FUNCTION_BLOCK "Side_Shifters"   // FB12, LAD
{ S7_Optimized_Access := 'TRUE' }
// stored: MemoryReserve 100, SetENOAutomatically false
   VAR_INPUT
      set_Hydraulic_Up { ExternalAccessible := 'False'; ExternalVisible := 'False'; ExternalWritable := 'False'} : Bool;
      set_Hydraulic_Down { ExternalAccessible := 'False'; ExternalVisible := 'False'; ExternalWritable := 'False'} : Bool;
      set_SL_Hydraulic_Up : Bool;
      set_SL_Hydraulic_Down : Bool;
      set_SR_Hydraulic_Up : Bool;
      set_SR_Hydraulic_Down : Bool;
      set_SL_Hydraulic_Unit : Bool;
      set_SR_Hydraulic_Unit : Bool;
      set_Go_To_ST1 : Bool;
      set_Go_To_ST2 : Bool;
      set_Go_To_ST3 : Bool;
      set_Go_To_ST4 : Bool;
      ST1_Empty : Bool;
      ST2_Empty : Bool;
      ST3_Empty : Bool;
      ST4_Empty : Bool;
      Homing_1_SR : Int;
      Homing_2_SR : Int;
      Homing_3_SR : Int;
      Homing_4_SR : Int;
      Homing_1_SL : Int;
      Homing_2_SL : Int;
      Homing_3_SL : Int;
      Homing_4_SL : Int;
      SL_Drive_Forward : Bool;
      SL_Drive_Backward : Bool;
      SR_Drive_Forward : Bool;
      SR_Drive_Backward : Bool;
      iSL_Sen_Drv_1 : Bool;
      iSL_Sen_Drv_2 : Bool;
      iSL_Sen_Drv_3 : Bool;
      iSL_Sen_Drv_4 : Bool;
      iSR_Sen_Drv_1 : Bool;
      iSR_Sen_Drv_2 : Bool;
      iSR_Sen_Drv_3 : Bool;
      iSR_Sen_Drv_4 : Bool;
      iSL_Sen_Val1_Up : Bool;
      iSL_Sen_Val1_Down : Bool;
      iSL_Sen_Val2_Up : Bool;
      iSL_Sen_Val2_Down : Bool;
      iSR_Sen_Val1_Up : Bool;
      iSR_Sen_Val1_Down : Bool;
      iSR_Sen_Val2_Up : Bool;
      iSR_Sen_Val2_Down : Bool;
      iSL_Distance : Int;
      iSR_Correct : Int;
      iSR_Distance : Int;
      iSL_Hydraulic_Filtr : Bool;
      iSR_Hydraulic_Empty : Bool;
      HWIdentSL : HW_IO;
      HWIdentSR : HW_IO;
      Reset_Drive : Bool;
      Reset_Hydro : Bool;
   END_VAR
   VAR_OUTPUT
      oSL_Valve_Up { ExternalAccessible := 'False'; ExternalVisible := 'False'; ExternalWritable := 'False'} : Bool;
      oSL_Valve_Down { ExternalAccessible := 'False'; ExternalVisible := 'False'; ExternalWritable := 'False'} : Bool;
      oSL_Hydraulic_Unit { ExternalAccessible := 'False'; ExternalVisible := 'False'; ExternalWritable := 'False'} : Bool;
      oSR_Valve_Up { ExternalAccessible := 'False'; ExternalVisible := 'False'; ExternalWritable := 'False'} : Bool;
      oSR_Valve_Down { ExternalAccessible := 'False'; ExternalVisible := 'False'; ExternalWritable := 'False'} : Bool;
      oSR_Hydraulic_Unit { ExternalAccessible := 'False'; ExternalVisible := 'False'; ExternalWritable := 'False'} : Bool;
      oHydraulic_Status_LED_UP_1 : Bool;
      oHydraulic_Status_LED_UP_2 : Bool;
      oHydraulic_Status_LED_DOWN_1 : Bool;
      oHydraulic_Status_LED_DOWN_2 : Bool;
      oSL_Communication_OK : Bool;
      oSR_Communication_OK : Bool;
      oSL_Forward_Flag : Bool;
      oSL_Backward_Flag : Bool;
      oSR_Forward_Flag : Bool;
      oSR_Backward_Flag : Bool;
      oST1_1_Move_Flag : Bool;
      oST1_2_Move_Flag : Bool;
      oST2_1_Move_Flag : Bool;
      oST2_2_Move_Flag : Bool;
      oST3_1_Move_flag : Bool;
      oST3_2_Move_Flag : Bool;
      oST4_1_Move_Flag : Bool;
      oST4_2_Move_Flag : Bool;
   END_VAR
   VAR_IN_OUT
      iSL_Drive_Param : "SEW_MOVIKIT_VelocityDrive_STATUS_V2.1";
      iSR_Drive_Param : "SEW_MOVIKIT_VelocityDrive_STATUS_V2.1";
      oSL_Drive_Param : "SEW_MOVIKIT_VelocityDrive_SETPOINTS_V2.1";
      oSR_Drive_Param : "SEW_MOVIKIT_VelocityDrive_SETPOINTS_V2.1";
   END_VAR
   VAR
      Hydraulic_SL { ExternalAccessible := 'False'; ExternalVisible := 'False'; ExternalWritable := 'False'} : "Side_Hydraulic";
      Hydraulic_SR { ExternalAccessible := 'False'; ExternalVisible := 'False'; ExternalWritable := 'False'} : "Side_Hydraulic";
      Side_Driver_Instance { S7_SetPoint := 'True'} : "Side_Driver";
      Side_Shifter_Auto_Instance { S7_SetPoint := 'True'} : "Side_Shifter_Auto";
      SL_Auto_Speed { S7_SetPoint := 'True'} : Int := 1000;
      SR_Auto_Speed { S7_SetPoint := 'True'} : Int := 1000;
      SL_Auto_Forward : Bool;
      SL_Auto_Backward : Bool;
      SR_Auto_Forward : Bool;
      SR_Auto_Backward : Bool;
      SR_Distance_Correct : Int;
      SL_Error_Laser : Bool;
      SR_Error_Laser : Bool;
      SL_SR_InPosition : Bool;
      SL_Sen_Up : Bool;
      SL_Sen_Down : Bool;
      SR_Sen_Up : Bool;
      SR_Sen_Down : Bool;
      SL_Error_Hyd : Bool;
      SR_Error_Hyd : Bool;
      Error_Drive : Bool;
      Error_Hydro : Bool;
      Status_Sen_Up : Bool;
      Status_Sen_Down : Bool;
      RL_Speed : Int;
      RR_Speed : Int;
      Step_Move_Pallets : Int;
      Row_Start : Int;
      Row_Destination : Int;
      Column_Start : Int;
      Column_Destination : Int;
      TON_iSR_Error { S7_SetPoint := 'True'} : TON_TIME;
      TON_iSL_Error { S7_SetPoint := 'True'} : TON_TIME;
   END_VAR
   VAR_TEMP
      i : SInt;
      FoundIndex : SInt;
   END_VAR
BEGIN

REGION Network 1: Hydraulic control SL
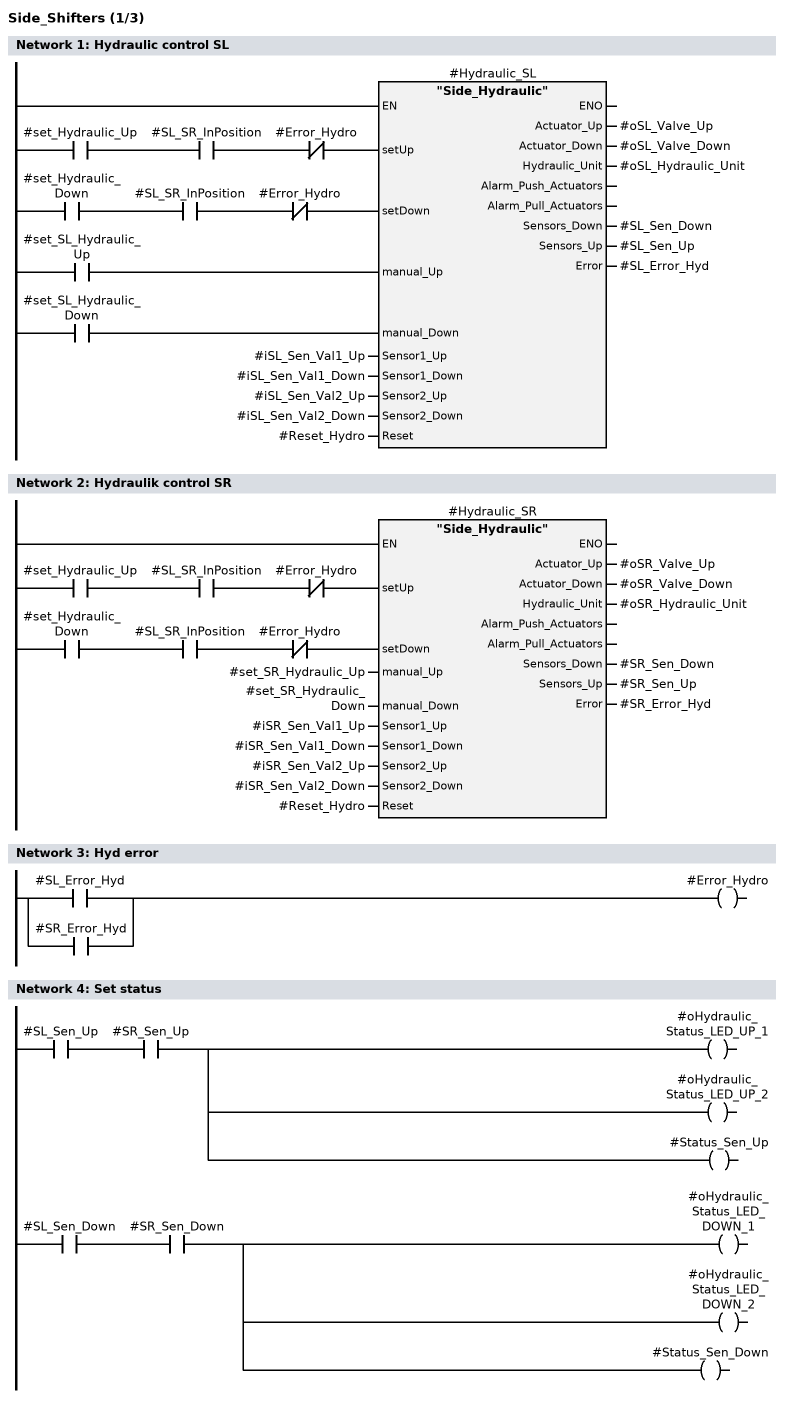
   RUNG wire#powerrail
      #Hydraulic_SL(setUp := wire#w1, setDown := wire#w2, manual_Up := wire#w3, manual_Down := wire#w4, Sensor1_Up := #iSL_Sen_Val1_Up, Sensor1_Down := #iSL_Sen_Val1_Down, Sensor2_Up := #iSL_Sen_Val2_Up, Sensor2_Down := #iSL_Sen_Val2_Down, Reset := #Reset_Hydro, Actuator_Up => #oSL_Valve_Up, Actuator_Down => #oSL_Valve_Down, Hydraulic_Unit => #oSL_Hydraulic_Unit, Alarm_Push_Actuators =>, Alarm_Pull_Actuators =>, Sensors_Down => #SL_Sen_Down, Sensors_Up => #SL_Sen_Up, Error => #SL_Error_Hyd)
   END_RUNG
   RUNG wire#powerrail
      Contact( #set_Hydraulic_Up )
      Contact( #SL_SR_InPosition )
      I_Contact( #Error_Hydro )
   END_RUNG wire#w1
   RUNG wire#powerrail
      Contact( #set_Hydraulic_Down )
      Contact( #SL_SR_InPosition )
      I_Contact( #Error_Hydro )
   END_RUNG wire#w2
   RUNG wire#powerrail
      Contact( #set_SL_Hydraulic_Up )
   END_RUNG wire#w3
   RUNG wire#powerrail
      Contact( #set_SL_Hydraulic_Down )
   END_RUNG wire#w4
   // the same network as SCL:
   #Hydraulic_SL(setUp := #set_Hydraulic_Up AND #SL_SR_InPosition AND NOT #Error_Hydro,   // "Side_Hydraulic"
                 setDown := #set_Hydraulic_Down AND #SL_SR_InPosition AND NOT #Error_Hydro,
                 manual_Up := #set_SL_Hydraulic_Up,
                 manual_Down := #set_SL_Hydraulic_Down,
                 Sensor1_Up := #iSL_Sen_Val1_Up,
                 Sensor1_Down := #iSL_Sen_Val1_Down,
                 Sensor2_Up := #iSL_Sen_Val2_Up,
                 Sensor2_Down := #iSL_Sen_Val2_Down,
                 Reset := #Reset_Hydro,
                 Actuator_Up => #oSL_Valve_Up,
                 Actuator_Down => #oSL_Valve_Down,
                 Hydraulic_Unit => #oSL_Hydraulic_Unit,
                 Sensors_Down => #SL_Sen_Down,
                 Sensors_Up => #SL_Sen_Up,
                 Error => #SL_Error_Hyd);
END_REGION

REGION Network 2: Hydraulik control SR
   RUNG wire#powerrail
      #Hydraulic_SR(setUp := wire#w1, setDown := wire#w2, manual_Up := #set_SR_Hydraulic_Up, manual_Down := #set_SR_Hydraulic_Down, Sensor1_Up := #iSR_Sen_Val1_Up, Sensor1_Down := #iSR_Sen_Val1_Down, Sensor2_Up := #iSR_Sen_Val2_Up, Sensor2_Down := #iSR_Sen_Val2_Down, Reset := #Reset_Hydro, Actuator_Up => #oSR_Valve_Up, Actuator_Down => #oSR_Valve_Down, Hydraulic_Unit => #oSR_Hydraulic_Unit, Alarm_Push_Actuators =>, Alarm_Pull_Actuators =>, Sensors_Down => #SR_Sen_Down, Sensors_Up => #SR_Sen_Up, Error => #SR_Error_Hyd)
   END_RUNG
   RUNG wire#powerrail
      Contact( #set_Hydraulic_Up )
      Contact( #SL_SR_InPosition )
      I_Contact( #Error_Hydro )
   END_RUNG wire#w1
   RUNG wire#powerrail
      Contact( #set_Hydraulic_Down )
      Contact( #SL_SR_InPosition )
      I_Contact( #Error_Hydro )
   END_RUNG wire#w2
   // the same network as SCL:
   #Hydraulic_SR(setUp := #set_Hydraulic_Up AND #SL_SR_InPosition AND NOT #Error_Hydro,   // "Side_Hydraulic"
                 setDown := #set_Hydraulic_Down AND #SL_SR_InPosition AND NOT #Error_Hydro,
                 manual_Up := #set_SR_Hydraulic_Up,
                 manual_Down := #set_SR_Hydraulic_Down,
                 Sensor1_Up := #iSR_Sen_Val1_Up,
                 Sensor1_Down := #iSR_Sen_Val1_Down,
                 Sensor2_Up := #iSR_Sen_Val2_Up,
                 Sensor2_Down := #iSR_Sen_Val2_Down,
                 Reset := #Reset_Hydro,
                 Actuator_Up => #oSR_Valve_Up,
                 Actuator_Down => #oSR_Valve_Down,
                 Hydraulic_Unit => #oSR_Hydraulic_Unit,
                 Sensors_Down => #SR_Sen_Down,
                 Sensors_Up => #SR_Sen_Up,
                 Error => #SR_Error_Hyd);
END_REGION

REGION Network 3: Hyd error
   RUNG wire#powerrail
      Contact( #SL_Error_Hyd )
      wire#w1
      Coil( #Error_Hydro )
   END_RUNG
   RUNG wire#powerrail
      Contact( #SR_Error_Hyd )
   END_RUNG wire#w1
   // the same network as SCL:
   #Error_Hydro := #SL_Error_Hyd OR #SR_Error_Hyd;
END_REGION

REGION Network 4: Set status
   RUNG wire#powerrail
      Contact( #SL_Sen_Up )
      Contact( #SR_Sen_Up )
      wire#w1
      Coil( #oHydraulic_Status_LED_UP_1 )
   END_RUNG
   RUNG wire#w1
      Coil( #oHydraulic_Status_LED_UP_2 )
   END_RUNG
   RUNG wire#w1
      Coil( #Status_Sen_Up )
   END_RUNG
   RUNG wire#powerrail
      Contact( #SL_Sen_Down )
      Contact( #SR_Sen_Down )
      wire#w2
      Coil( #oHydraulic_Status_LED_DOWN_1 )
   END_RUNG
   RUNG wire#w2
      Coil( #oHydraulic_Status_LED_DOWN_2 )
   END_RUNG
   RUNG wire#w2
      Coil( #Status_Sen_Down )
   END_RUNG
   // the same network as SCL:
   #oHydraulic_Status_LED_UP_1 := #SL_Sen_Up AND #SR_Sen_Up;
   #oHydraulic_Status_LED_UP_2 := #oHydraulic_Status_LED_UP_1;
   #Status_Sen_Up := #oHydraulic_Status_LED_UP_1;
   #oHydraulic_Status_LED_DOWN_1 := #SL_Sen_Down AND #SR_Sen_Down;
   #oHydraulic_Status_LED_DOWN_2 := #oHydraulic_Status_LED_DOWN_1;
   #Status_Sen_Down := #oHydraulic_Status_LED_DOWN_1;
END_REGION

REGION Network 5: Make correct on SR distance
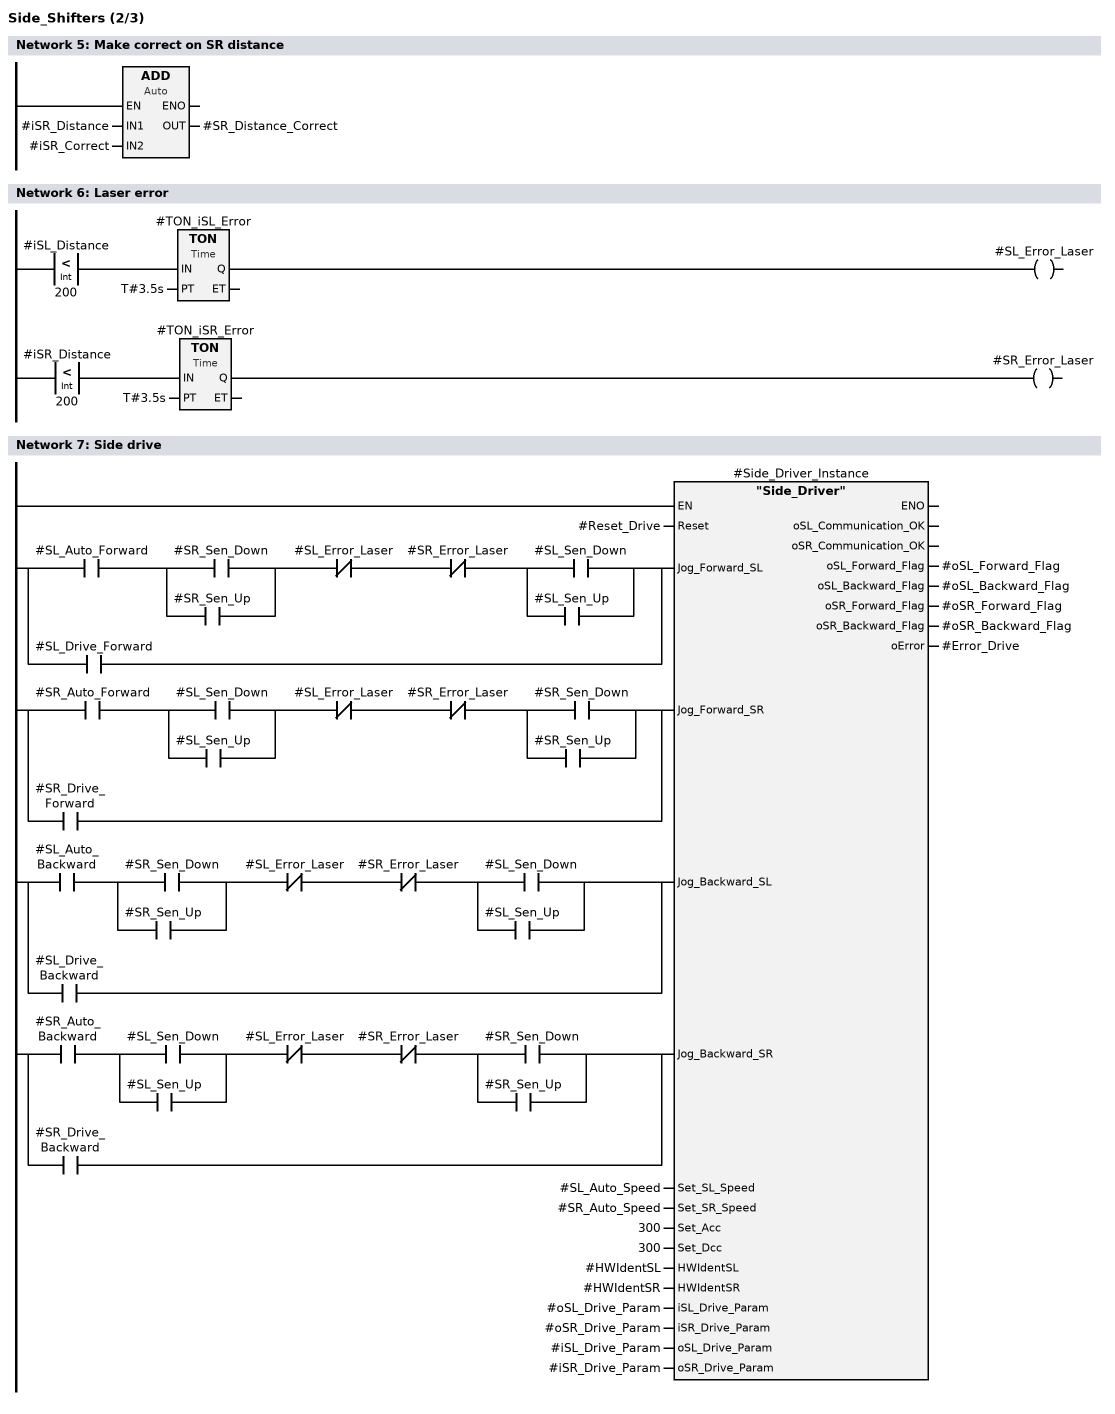
   RUNG wire#powerrail
      Add(in1 := #iSR_Distance, in2 := #iSR_Correct, out => #SR_Distance_Correct)
   END_RUNG
   // the same network as SCL:
   #SR_Distance_Correct := #iSR_Distance + #iSR_Correct;
END_REGION

REGION Network 6: Laser error
   RUNG wire#powerrail
      { S7_Templates := "SrcType := Int" } LT_Contact(in1 := #iSL_Distance, in2 := 200)
      { S7_Templates := "time_type := Time" } #TON_iSL_Error.TON(pt := T#3.5s, et =>)
      Coil( #SL_Error_Laser )
   END_RUNG
   RUNG wire#powerrail
      { S7_Templates := "SrcType := Int" } LT_Contact(in1 := #iSR_Distance, in2 := 200)
      { S7_Templates := "time_type := Time" } #TON_iSR_Error.TON(pt := T#3.5s, et =>)
      Coil( #SR_Error_Laser )
   END_RUNG
   // the same network as SCL:
   #TON_iSL_Error(IN := #iSL_Distance < 200, PT := T#3.5s);   // TON
   #SL_Error_Laser := #TON_iSL_Error.Q;
   #TON_iSR_Error(IN := #iSR_Distance < 200, PT := T#3.5s);   // TON
   #SR_Error_Laser := #TON_iSR_Error.Q;
END_REGION

REGION Network 7: Side drive
   RUNG wire#powerrail
      #Side_Driver_Instance(Jog_Forward_SL := wire#w4, Jog_Forward_SR := wire#w8, Jog_Backward_SL := wire#w12, Jog_Backward_SR := wire#w16, Reset := #Reset_Drive, Set_SL_Speed := #SL_Auto_Speed, Set_SR_Speed := #SR_Auto_Speed, Set_Acc := 300, Set_Dcc := 300, HWIdentSL := #HWIdentSL, HWIdentSR := #HWIdentSR, iSL_Drive_Param := #oSL_Drive_Param, iSR_Drive_Param := #oSR_Drive_Param, oSL_Drive_Param := #iSL_Drive_Param, oSR_Drive_Param := #iSR_Drive_Param, oSL_Communication_OK =>, oSR_Communication_OK =>, oSL_Forward_Flag => #oSL_Forward_Flag, oSL_Backward_Flag => #oSL_Backward_Flag, oSR_Forward_Flag => #oSR_Forward_Flag, oSR_Backward_Flag => #oSR_Backward_Flag, oError => #Error_Drive)
   END_RUNG
   RUNG wire#powerrail
      Contact( #SL_Auto_Forward )
      wire#w1
      Contact( #SR_Sen_Down )
      wire#w2
      I_Contact( #SL_Error_Laser )
      I_Contact( #SR_Error_Laser )
      wire#w3
      Contact( #SL_Sen_Down )
   END_RUNG wire#w4
   RUNG wire#w1
      Contact( #SR_Sen_Up )
   END_RUNG wire#w2
   RUNG wire#w3
      Contact( #SL_Sen_Up )
   END_RUNG wire#w4
   RUNG wire#powerrail
      Contact( #SL_Drive_Forward )
   END_RUNG wire#w4
   RUNG wire#powerrail
      Contact( #SR_Auto_Forward )
      wire#w5
      Contact( #SL_Sen_Down )
      wire#w6
      I_Contact( #SL_Error_Laser )
      I_Contact( #SR_Error_Laser )
      wire#w7
      Contact( #SR_Sen_Down )
   END_RUNG wire#w8
   RUNG wire#w5
      Contact( #SL_Sen_Up )
   END_RUNG wire#w6
   RUNG wire#w7
      Contact( #SR_Sen_Up )
   END_RUNG wire#w8
   RUNG wire#powerrail
      Contact( #SR_Drive_Forward )
   END_RUNG wire#w8
   RUNG wire#powerrail
      Contact( #SL_Auto_Backward )
      wire#w9
      Contact( #SR_Sen_Down )
      wire#w10
      I_Contact( #SL_Error_Laser )
      I_Contact( #SR_Error_Laser )
      wire#w11
      Contact( #SL_Sen_Down )
   END_RUNG wire#w12
   RUNG wire#w9
      Contact( #SR_Sen_Up )
   END_RUNG wire#w10
   RUNG wire#w11
      Contact( #SL_Sen_Up )
   END_RUNG wire#w12
   RUNG wire#powerrail
      Contact( #SL_Drive_Backward )
   END_RUNG wire#w12
   RUNG wire#powerrail
      Contact( #SR_Auto_Backward )
      wire#w13
      Contact( #SL_Sen_Down )
      wire#w14
      I_Contact( #SL_Error_Laser )
      I_Contact( #SR_Error_Laser )
      wire#w15
      Contact( #SR_Sen_Down )
   END_RUNG wire#w16
   RUNG wire#w13
      Contact( #SL_Sen_Up )
   END_RUNG wire#w14
   RUNG wire#w15
      Contact( #SR_Sen_Up )
   END_RUNG wire#w16
   RUNG wire#powerrail
      Contact( #SR_Drive_Backward )
   END_RUNG wire#w16
   // the same network as SCL:
   #Side_Driver_Instance(Reset := #Reset_Drive,   // "Side_Driver"
                         Jog_Forward_SL := (#SL_Auto_Forward AND (#SR_Sen_Down OR #SR_Sen_Up) AND NOT #SL_Error_Laser AND NOT #SR_Error_Laser AND (#SL_Sen_Down OR #SL_Sen_Up)) OR #SL_Drive_Forward,
                         Jog_Forward_SR := (#SR_Auto_Forward AND (#SL_Sen_Down OR #SL_Sen_Up) AND NOT #SL_Error_Laser AND NOT #SR_Error_Laser AND (#SR_Sen_Down OR #SR_Sen_Up)) OR #SR_Drive_Forward,
                         Jog_Backward_SL := (#SL_Auto_Backward AND (#SR_Sen_Down OR #SR_Sen_Up) AND NOT #SL_Error_Laser AND NOT #SR_Error_Laser AND (#SL_Sen_Down OR #SL_Sen_Up)) OR #SL_Drive_Backward,
                         Jog_Backward_SR := (#SR_Auto_Backward AND (#SL_Sen_Down OR #SL_Sen_Up) AND NOT #SL_Error_Laser AND NOT #SR_Error_Laser AND (#SR_Sen_Down OR #SR_Sen_Up)) OR #SR_Drive_Backward,
                         Set_SL_Speed := #SL_Auto_Speed,
                         Set_SR_Speed := #SR_Auto_Speed,
                         Set_Acc := 300,
                         Set_Dcc := 300,
                         HWIdentSL := #HWIdentSL,
                         HWIdentSR := #HWIdentSR,
                         iSL_Drive_Param := #oSL_Drive_Param,
                         iSR_Drive_Param := #oSR_Drive_Param,
                         oSL_Drive_Param := #iSL_Drive_Param,
                         oSR_Drive_Param := #iSR_Drive_Param,
                         oSL_Forward_Flag => #oSL_Forward_Flag,
                         oSL_Backward_Flag => #oSL_Backward_Flag,
                         oSR_Forward_Flag => #oSR_Forward_Flag,
                         oSR_Backward_Flag => #oSR_Backward_Flag,
                         oError => #Error_Drive);
END_REGION

REGION Network 8: Auto moving
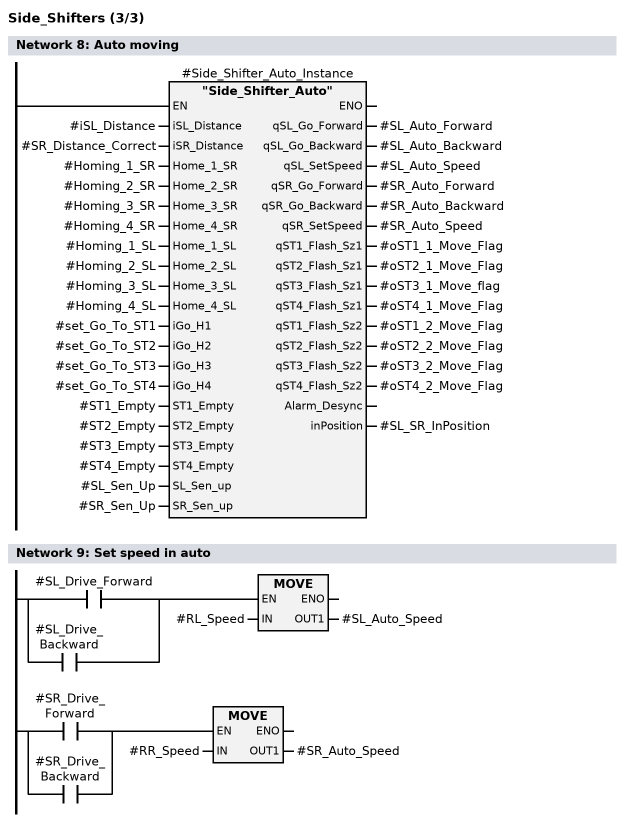
   RUNG wire#powerrail
      #Side_Shifter_Auto_Instance(iSL_Distance := #iSL_Distance, iSR_Distance := #SR_Distance_Correct, Home_1_SR := #Homing_1_SR, Home_2_SR := #Homing_2_SR, Home_3_SR := #Homing_3_SR, Home_4_SR := #Homing_4_SR, Home_1_SL := #Homing_1_SL, Home_2_SL := #Homing_2_SL, Home_3_SL := #Homing_3_SL, Home_4_SL := #Homing_4_SL, iGo_H1 := #set_Go_To_ST1, iGo_H2 := #set_Go_To_ST2, iGo_H3 := #set_Go_To_ST3, iGo_H4 := #set_Go_To_ST4, ST1_Empty := #ST1_Empty, ST2_Empty := #ST2_Empty, ST3_Empty := #ST3_Empty, ST4_Empty := #ST4_Empty, SL_Sen_up := #SL_Sen_Up, SR_Sen_up := #SR_Sen_Up, qSL_Go_Forward => #SL_Auto_Forward, qSL_Go_Backward => #SL_Auto_Backward, qSL_SetSpeed => #SL_Auto_Speed, qSR_Go_Forward => #SR_Auto_Forward, qSR_Go_Backward => #SR_Auto_Backward, qSR_SetSpeed => #SR_Auto_Speed, qST1_Flash_Sz1 => #oST1_1_Move_Flag, qST2_Flash_Sz1 => #oST2_1_Move_Flag, qST3_Flash_Sz1 => #oST3_1_Move_flag, qST4_Flash_Sz1 => #oST4_1_Move_Flag, qST1_Flash_Sz2 => #oST1_2_Move_Flag, qST2_Flash_Sz2 => #oST2_2_Move_Flag, qST3_Flash_Sz2 => #oST3_2_Move_Flag, qST4_Flash_Sz2 => #oST4_2_Move_Flag, Alarm_Desync =>, inPosition => #SL_SR_InPosition)
   END_RUNG
   // the same network as SCL:
   #Side_Shifter_Auto_Instance(iSL_Distance := #iSL_Distance,   // "Side_Shifter_Auto"
                           iSR_Distance := #SR_Distance_Correct,
                           Home_1_SR := #Homing_1_SR,
                           Home_2_SR := #Homing_2_SR,
                           Home_3_SR := #Homing_3_SR,
                           Home_4_SR := #Homing_4_SR,
                           Home_1_SL := #Homing_1_SL,
                           Home_2_SL := #Homing_2_SL,
                           Home_3_SL := #Homing_3_SL,
                           Home_4_SL := #Homing_4_SL,
                           iGo_H1 := #set_Go_To_ST1,
                           iGo_H2 := #set_Go_To_ST2,
                           iGo_H3 := #set_Go_To_ST3,
                           iGo_H4 := #set_Go_To_ST4,
                           ST1_Empty := #ST1_Empty,
                           ST2_Empty := #ST2_Empty,
                           ST3_Empty := #ST3_Empty,
                           ST4_Empty := #ST4_Empty,
                           SL_Sen_up := #SL_Sen_Up,
                           SR_Sen_up := #SR_Sen_Up,
                           qSL_Go_Forward => #SL_Auto_Forward,
                           qSL_Go_Backward => #SL_Auto_Backward,
                           qSL_SetSpeed => #SL_Auto_Speed,
                           qSR_Go_Forward => #SR_Auto_Forward,
                           qSR_Go_Backward => #SR_Auto_Backward,
                           qSR_SetSpeed => #SR_Auto_Speed,
                           qST1_Flash_Sz1 => #oST1_1_Move_Flag,
                           qST2_Flash_Sz1 => #oST2_1_Move_Flag,
                           qST3_Flash_Sz1 => #oST3_1_Move_flag,
                           qST4_Flash_Sz1 => #oST4_1_Move_Flag,
                           qST1_Flash_Sz2 => #oST1_2_Move_Flag,
                           qST2_Flash_Sz2 => #oST2_2_Move_Flag,
                           qST3_Flash_Sz2 => #oST3_2_Move_Flag,
                           qST4_Flash_Sz2 => #oST4_2_Move_Flag,
                           inPosition => #SL_SR_InPosition);
END_REGION

REGION Network 9: Set speed in auto
   RUNG wire#powerrail
      Contact( #SL_Drive_Forward )
      wire#w1
      Move(in := #RL_Speed, out1 => #SL_Auto_Speed)
   END_RUNG
   RUNG wire#powerrail
      Contact( #SL_Drive_Backward )
   END_RUNG wire#w1
   RUNG wire#powerrail
      Contact( #SR_Drive_Forward )
      wire#w2
      Move(in := #RR_Speed, out1 => #SR_Auto_Speed)
   END_RUNG
   RUNG wire#powerrail
      Contact( #SR_Drive_Backward )
   END_RUNG wire#w2
   // the same network as SCL:
   IF #SL_Drive_Forward OR #SL_Drive_Backward THEN #SL_Auto_Speed := #RL_Speed; END_IF;
   IF #SR_Drive_Forward OR #SR_Drive_Backward THEN #SR_Auto_Speed := #RR_Speed; END_IF;
END_REGION

REGION Network 10 (SCL): SS1 - Move Pallet
   IF #HWIdentSL = "S1R1M~Module_I_O_(05_words)_1" THEN

       IF (#Hydraulic_SL.Actuator_Up OR #Hydraulic_SR.Actuator_Up) AND #Status_Sen_Up AND #Step_Move_Pallets = 0 THEN
           #Step_Move_Pallets := 1;
           IF #oST1_1_Move_Flag THEN
               #Row_Start := 1;
               #Column_Start := 11;
           ELSIF #oST2_1_Move_Flag THEN
               #Row_Start := 2;
               #Column_Start := 12;
           ELSIF #oST3_1_Move_flag THEN
               #Row_Start := 3;
               #Column_Start := 11;
           ELSIF #oST4_1_Move_Flag THEN
               #Row_Start := 4;
               #Column_Start := 11;
           END_IF;

       ELSIF (#Hydraulic_SL.Actuator_Down OR #Hydraulic_SR.Actuator_Down) AND #Status_Sen_Up AND #Step_Move_Pallets = 1 THEN
           #Step_Move_Pallets := 2;
           IF #oST1_1_Move_Flag THEN
               #Row_Destination := 1;
               #Column_Destination := 11;
           ELSIF #oST2_1_Move_Flag THEN
               #Row_Destination := 2;
               #Column_Destination := 12;
           ELSIF #oST3_1_Move_flag THEN
               #Row_Destination := 3;
               #Column_Destination := 11;
           ELSIF #oST4_1_Move_Flag THEN
               #Row_Destination := 4;
               #Column_Destination := 11;
           END_IF;

       ELSIF #Step_Move_Pallets = 2 THEN
           FOR #i := 1 TO 24 DO
               IF ("Pallets_Stations".Pallets[#i].Station_Current_Position[1] = #Row_Start) AND
                   ("Pallets_Stations".Pallets[#i].Station_Current_Position[2] = #Column_Start) THEN
                   #FoundIndex := #i;
                   EXIT;
               END_IF;
           END_FOR;

           IF #FoundIndex <> 0 THEN
               "Pallets_Stations".Pallets[#FoundIndex].Station_Current_Position[1] := #Row_Destination;
               "Pallets_Stations".Pallets[#FoundIndex].Station_Current_Position[2] := #Column_Destination;
           END_IF;
           #Step_Move_Pallets := 0;

       END_IF;
   END_IF;
END_REGION

REGION Network 11 (SCL): SS2 - Move Pallet
   IF #HWIdentSL = "S2R2M~Module_I_O_(05_words)_1" THEN
       #Column_Start := 1;
       IF (#Hydraulic_SL.Actuator_Up OR #Hydraulic_SR.Actuator_Up) AND #Status_Sen_Up AND #Step_Move_Pallets = 0 THEN
           #Step_Move_Pallets := 1;
           IF #oST1_1_Move_Flag THEN
               #Row_Start := 1;
           ELSIF #oST2_1_Move_Flag THEN
               #Row_Start := 2;
           ELSIF #oST3_1_Move_flag THEN
               #Row_Start := 3;
           ELSIF #oST4_1_Move_Flag THEN
               #Row_Start := 4;
           END_IF;

       ELSIF (#Hydraulic_SL.Actuator_Down OR #Hydraulic_SR.Actuator_Down) AND #Status_Sen_Up AND #Step_Move_Pallets = 1 THEN
           #Step_Move_Pallets := 2;
           IF #oST1_1_Move_Flag THEN
               #Row_Destination := 1;
           ELSIF #oST2_1_Move_Flag THEN
               #Row_Destination := 2;
           ELSIF #oST3_1_Move_flag THEN
               #Row_Destination := 3;
           ELSIF #oST4_1_Move_Flag THEN
               #Row_Destination := 4;
           END_IF;

       ELSIF #Step_Move_Pallets = 2 THEN
           FOR #i := 1 TO 24 DO
               IF ("Pallets_Stations".Pallets[#i].Station_Current_Position[1] = #Row_Start) AND
                   ("Pallets_Stations".Pallets[#i].Station_Current_Position[2] = #Column_Start) THEN
                   #FoundIndex := #i;
                   EXIT;
               END_IF;
           END_FOR;

           IF #FoundIndex <> 0 THEN
               "Pallets_Stations".Pallets[#FoundIndex].Station_Current_Position[1] := #Row_Destination;
               "Pallets_Stations".Pallets[#FoundIndex].Station_Current_Position[2] := #Column_Destination;
           END_IF;
           #Step_Move_Pallets := 0;

       END_IF;
   END_IF;
END_REGION
END_FUNCTION_BLOCK

FUNCTION_BLOCK "Side_Shifter_Auto"   // FB13, LAD
{ S7_Optimized_Access := 'TRUE' }
// stored: MemoryReserve 100, SetENOAutomatically false
   VAR_INPUT
      iSL_Distance : Int;
      iSR_Distance : Int;
      Home_1_SR : Int;
      Home_2_SR : Int;
      Home_3_SR : Int;
      Home_4_SR : Int;
      Home_1_SL : Int;
      Home_2_SL : Int;
      Home_3_SL : Int;
      Home_4_SL : Int;
      iGo_H1 : Bool;
      iGo_H2 : Bool;
      iGo_H3 : Bool;
      iGo_H4 : Bool;
      ST1_Empty : Bool;
      ST2_Empty : Bool;
      ST3_Empty : Bool;
      ST4_Empty : Bool;
      SL_Sen_up : Bool;
      SR_Sen_up : Bool;
   END_VAR
   VAR_OUTPUT
      qSL_Go_Forward : Bool;
      qSL_Go_Backward : Bool;
      qSL_SetSpeed : Int;
      qSR_Go_Forward : Bool;
      qSR_Go_Backward : Bool;
      qSR_SetSpeed : Int;
      qST1_Flash_Sz1 : Bool;
      qST2_Flash_Sz1 : Bool;
      qST3_Flash_Sz1 : Bool;
      qST4_Flash_Sz1 : Bool;
      qST1_Flash_Sz2 : Bool := false;
      qST2_Flash_Sz2 : Bool := false;
      qST3_Flash_Sz2 : Bool := false;
      qST4_Flash_Sz2 : Bool := false;
      Alarm_Desync : Bool;
      inPosition : Bool;
   END_VAR
   VAR
      targetPosSR : Int;
      targetPosSL : Int;
      moveActive : Bool;
      distanceToTargetSL : Int;
      distanceToTargetSR : Int;
      distanceSL_SR : Int;
      selectedStation : Int;
      maxDelta : Real;
      k_sync : Real;
      deltaClamped : Real;
      Delta : Real;
      moveActive_SL : Bool;
      moveActive_SR : Bool;
      distanceToTarget_SL : Int;
      distanceToTarget_SR : Int;
      NominalOffset : Int;
      syncError : Int;
      baseSpeedSR : Real;
      sensorErrorTimer : TON_TIME;
      pathClear { S7_SetPoint := 'True'} : Bool;
   END_VAR
   VAR_TEMP
      sensorErrorSL : Bool;
      sensorErrorSR : Bool;
      sensorErrorAny : Bool;
      sensorFallback : Bool;
   END_VAR
   VAR CONSTANT
      Tolerance : Int := 3;
      Tolerance_Light : Int := 5;
      Tolerance_Hydro : Int := 15;
      DistanceSlowZone : Int := 600;
      SpeedFast : Int := 1100;
      SpeedSlow : Int := 320;
      K : Real := 1.5;
      MaxOffset : Int := 200;
   END_VAR
BEGIN

REGION Network 1 (SCL)
   // RESET WYJŚĆ

   #qSL_Go_Forward := FALSE;
   #qSL_Go_Backward := FALSE;
   #qSR_Go_Forward := FALSE;
   #qSR_Go_Backward := FALSE;
   #qSL_SetSpeed := 0;
   #qSR_SetSpeed := 0;
   #Alarm_Desync := FALSE;

   // WYBÓR CELU

   IF #iGo_H1 THEN
       #targetPosSL := #Home_1_SL;
       #targetPosSR := #Home_1_SR;
       #moveActive := TRUE;

   ELSIF #iGo_H2 THEN
       #targetPosSL := #Home_2_SL;
       #targetPosSR := #Home_2_SR;
       #moveActive := TRUE;

   ELSIF #iGo_H3 THEN
       #targetPosSL := #Home_3_SL;
       #targetPosSR := #Home_3_SR;
       #moveActive := TRUE;

   ELSIF #iGo_H4 THEN
       #targetPosSL := #Home_4_SL;
       #targetPosSR := #Home_4_SR;
       #moveActive := TRUE;

   ELSE
       #moveActive := FALSE;
   END_IF;

   // SAFETY

   IF NOT "Data_From_Safety".Safety_Active THEN
       #moveActive := FALSE;
   END_IF;

   // RUCH AKTYWNY

   IF #moveActive THEN

       // DETEKCJA BŁĘDU CZUJNIKÓW

       #sensorErrorSL := (#iSL_Distance < 100);
       #sensorErrorSR := (#iSR_Distance < 100);
       #sensorErrorAny := #sensorErrorSL OR #sensorErrorSR;

       #sensorErrorTimer(
                        IN := #sensorErrorAny,
                        PT := T#3s
       );

       // fallback tylko gdy padł JEDEN czujnik
       #sensorFallback :=
       (#sensorErrorSL XOR #sensorErrorSR)
       AND NOT #sensorErrorTimer.Q;


       // DISTANCE (tylko jeśli czujnik OK)

       IF NOT #sensorErrorSL THEN
           #distanceToTargetSL := ABS(#iSL_Distance - #targetPosSL);
       ELSE
           #distanceToTargetSL := 0;
       END_IF;

       IF NOT #sensorErrorSR THEN
           #distanceToTargetSR := ABS(#iSR_Distance - #targetPosSR);
       ELSE
           #distanceToTargetSR := 0;
       END_IF;


       // SL – KIERUNEK I PRĘDKOŚĆ

       IF NOT #sensorErrorSL AND (#distanceToTargetSL > #Tolerance) THEN

           IF #iSL_Distance > #targetPosSL THEN
               #qSL_Go_Forward := TRUE;
           ELSE
               #qSL_Go_Backward := TRUE;
           END_IF;

           IF #distanceToTargetSL <= #DistanceSlowZone THEN
               #qSL_SetSpeed := #SpeedSlow;
           ELSE
               #qSL_SetSpeed := #SpeedFast;
           END_IF;
       ELSE

           // DOJECHAŁ
           #qSL_SetSpeed := 0;
           #qSL_Go_Forward := FALSE;
           #qSL_Go_Backward := FALSE;
       END_IF;



       // SR – KIERUNEK I PRĘDKOŚĆ BAZOWA

       IF NOT #sensorErrorSR AND (#distanceToTargetSR > #Tolerance) THEN

           IF #iSR_Distance > #targetPosSR THEN
               #qSR_Go_Forward := TRUE;
           ELSE
               #qSR_Go_Backward := TRUE;
           END_IF;

           IF #distanceToTargetSR <= #DistanceSlowZone THEN
               #baseSpeedSR := #SpeedSlow;
           ELSE
               #baseSpeedSR := #SpeedFast;
           END_IF;
           #qSR_SetSpeed := #baseSpeedSR;;

       ELSE
           #qSR_SetSpeed := 0;
           #qSR_Go_Forward := FALSE;
           #qSR_Go_Backward := FALSE;
       END_IF;

       // SPRAWDZ KOLIZJE PRZY PRZEJEZDZIE DLA SL

       #pathClear := TRUE;

       IF #qSL_Go_Forward THEN

           IF ((#Home_1_SL < (#iSL_Distance - #Tolerance_Hydro)) AND (#Home_1_SL > #targetPosSL) AND NOT #ST1_Empty)
               OR ((#Home_2_SL < (#iSL_Distance - #Tolerance_Hydro)) AND (#Home_2_SL > #targetPosSL) AND NOT #ST2_Empty)
               OR ((#Home_3_SL < (#iSL_Distance - #Tolerance_Hydro)) AND (#Home_3_SL > #targetPosSL) AND NOT #ST3_Empty)
               OR ((#Home_4_SL < (#iSL_Distance - #Tolerance_Hydro)) AND (#Home_4_SL > #targetPosSL) AND NOT #ST4_Empty) THEN

               #pathClear := FALSE;

           END_IF;

       END_IF;



       IF #qSL_Go_Backward THEN

           IF ((#Home_1_SL > (#iSL_Distance + #Tolerance_Hydro)) AND (#Home_1_SL < #targetPosSL) AND NOT #ST1_Empty)
               OR ((#Home_2_SL > (#iSL_Distance + #Tolerance_Hydro)) AND (#Home_2_SL < #targetPosSL) AND NOT #ST2_Empty)
               OR ((#Home_3_SL > (#iSL_Distance + #Tolerance_Hydro)) AND (#Home_3_SL < #targetPosSL) AND NOT #ST3_Empty)
               OR ((#Home_4_SL > (#iSL_Distance + #Tolerance_Hydro)) AND (#Home_4_SL < #targetPosSL) AND NOT #ST4_Empty) THEN

               #pathClear := FALSE;

           END_IF;

       END_IF;

       // SYNCHRONIZACJA (TYLKO BEZ FALLBACKU)

       IF NOT #sensorFallback AND (#distanceToTargetSL > #Tolerance) AND (#distanceToTargetSR > #Tolerance) THEN

           #NominalOffset := #targetPosSR - #targetPosSL;
           #syncError := (#iSR_Distance - #iSL_Distance) - #NominalOffset;

           IF ABS(#syncError) > #MaxOffset THEN
               #qSL_Go_Forward := FALSE;
               #qSL_Go_Backward := FALSE;
               #qSR_Go_Forward := FALSE;
               #qSR_Go_Backward := FALSE;
               #qSL_SetSpeed := 0;
               #qSR_SetSpeed := 0;
               #Alarm_Desync := TRUE;
               #moveActive := FALSE;
           END_IF;

           #Delta := #syncError * #k_sync;

           IF #Delta > 300 THEN
               #Delta := 300;
           ELSIF #Delta < -300 THEN
               #Delta := -300;
           END_IF;

           #qSR_SetSpeed := #baseSpeedSR - #Delta;

           IF #qSR_SetSpeed > 1500 THEN
               #qSR_SetSpeed := 1500;
           ELSIF #qSR_SetSpeed < 200 AND #qSR_SetSpeed > 0 THEN
               #qSR_SetSpeed := 200;
           END_IF;

       END_IF;

       // FALLBACK – DWUKIERUNKOWY

       IF #sensorFallback THEN

           // SR padł → SR kopiuje SL
           IF #sensorErrorSR THEN
               #qSR_SetSpeed := #qSL_SetSpeed;
               #qSR_Go_Forward := #qSL_Go_Forward;
               #qSR_Go_Backward := #qSL_Go_Backward;
           END_IF;

           // SL padł → SL kopiuje SR
           IF #sensorErrorSL THEN
               #qSL_SetSpeed := #qSR_SetSpeed;
               #qSL_Go_Forward := #qSR_Go_Forward;
               #qSL_Go_Backward := #qSR_Go_Backward;
           END_IF;

       END_IF;

       // STOP JEŚLI BŁĄD > time

       IF #sensorErrorTimer.Q THEN
           #qSL_Go_Forward := FALSE;
           #qSL_Go_Backward := FALSE;
           #qSR_Go_Forward := FALSE;
           #qSR_Go_Backward := FALSE;
           #qSL_SetSpeed := 0;
           #qSR_SetSpeed := 0;
           #Alarm_Desync := TRUE;
           #moveActive := FALSE;
       END_IF;

       // ZAKOŃCZENIE RUCHU

       IF (NOT #sensorErrorSL) AND (NOT #sensorErrorSR) THEN
           IF (#distanceToTargetSL <= #Tolerance)
               AND (#distanceToTargetSR <= #Tolerance) THEN
               #moveActive := FALSE;
           END_IF;
       END_IF;

   END_IF;

   //BLOKUJ RUCH JESLI KOLIZJA
   IF NOT #pathClear AND #SR_Sen_up AND #SL_Sen_up THEN

       #qSL_Go_Forward := FALSE;
       #qSL_Go_Backward := FALSE;
       #qSR_Go_Forward := FALSE;
       #qSR_Go_Backward := FALSE;

       #qSL_SetSpeed := 0;
       #qSR_SetSpeed := 0;

       #moveActive := FALSE;

   END_IF;


   // IN POSITION

   #inPosition :=
   (NOT #sensorErrorSL) AND (NOT #sensorErrorSR)
   AND (ABS(#iSL_Distance - #targetPosSL) <= #Tolerance_Hydro)
   AND (ABS(#iSR_Distance - #targetPosSR) <= #Tolerance_Hydro);

   // MIGANIE LAMPEK – PRZYCISK TRZYMANY + RUCH

   IF #moveActive AND "Clock_2Hz" THEN

       #qST1_Flash_Sz1 := #iGo_H1;
       #qST1_Flash_Sz2 := #iGo_H1;

       #qST2_Flash_Sz1 := #iGo_H2;
       #qST2_Flash_Sz2 := #iGo_H2;

       #qST3_Flash_Sz1 := #iGo_H3;
       #qST3_Flash_Sz2 := #iGo_H3;

       #qST4_Flash_Sz1 := #iGo_H4;
       #qST4_Flash_Sz2 := #iGo_H4;

   ELSE
       #qST1_Flash_Sz1 := 0;
       #qST1_Flash_Sz2 := 0;
       #qST2_Flash_Sz1 := 0;
       #qST2_Flash_Sz2 := 0;
       #qST3_Flash_Sz1 := 0;
       #qST3_Flash_Sz2 := 0;
       #qST4_Flash_Sz1 := 0;
       #qST4_Flash_Sz2 := 0;
   END_IF;

   // LAMPKI – DOJECHANO DO POZYCJI

   IF #inPosition THEN
       IF ABS(#iSL_Distance - #Home_1_SL) <= #Tolerance_Light
           AND ABS(#iSR_Distance - #Home_1_SR) <= #Tolerance_Light THEN
           #qST1_Flash_Sz1 := 1;
           #qST1_Flash_Sz2 := 1;

       ELSIF ABS(#iSL_Distance - #Home_2_SL) <= #Tolerance_Light
           AND ABS(#iSR_Distance - #Home_2_SR) <= #Tolerance_Light THEN
           #qST2_Flash_Sz1 := 1;
           #qST2_Flash_Sz2 := 1;

       ELSIF ABS(#iSL_Distance - #Home_3_SL) <= #Tolerance_Light
           AND ABS(#iSR_Distance - #Home_3_SR) <= #Tolerance_Light THEN
           #qST3_Flash_Sz1 := 1;
           #qST3_Flash_Sz2 := 1;

       ELSIF ABS(#iSL_Distance - #Home_4_SL) <= #Tolerance_Light
           AND ABS(#iSR_Distance - #Home_4_SR) <= #Tolerance_Light THEN
           #qST4_Flash_Sz1 := 1;
           #qST4_Flash_Sz2 := 1;
       END_IF;
   END_IF;
END_REGION
END_FUNCTION_BLOCK

FUNCTION_BLOCK "System_To_Moving_Pallets"   // FB15, LAD
{ S7_Optimized_Access := 'TRUE' }
// stored: MemoryReserve 100, SetENOAutomatically false
   VAR
      iCenterTippler : Bool;
      oCeterTippler : Bool;
      Reset_Centering_Tippler : Bool;
      ST13_ST14 { S7_SetPoint := 'True'} : "Pallet_Transport_Row_4";
      ST12_ST13 { S7_SetPoint := 'True'} : "Pallet_Transport_Row_4";
      ST11_ST12 { S7_SetPoint := 'True'} : "Pallet_Transport_Row_4";
      ST10_ST11 { S7_SetPoint := 'True'} : "Pallet_Transport_Row_4";
      ST09_ST10 { S7_SetPoint := 'True'} : "Pallet_Transport_Row_4";
      ST08_ST09 { S7_SetPoint := 'True'} : "Pallet_Transport_Row_4";
      ST07_ST08 { S7_SetPoint := 'True'} : "Pallet_Transport_Row_4";
      ST06_ST07 { S7_SetPoint := 'True'} : "Pallet_Transport_Row_4";
      ST05_ST06 { S7_SetPoint := 'True'} : "Pallet_Transport_Row_4";
      ST04_ST05 { S7_SetPoint := 'True'} : "Pallet_Transport_Row_4";
      ST01_ST02 { S7_SetPoint := 'True'} : "Pallet_Transport_Row_1_2";
      ST02_ST01 { S7_SetPoint := 'True'} : "Pallet_Transport_Row_1_2";
      ST38_ST01 { S7_SetPoint := 'True'} : "Pallet_Transport_Row_1_2";
      ST01_ST38 { S7_SetPoint := 'True'} : "Pallet_Transport_Row_1_2";
      ST34_ST35 { S7_SetPoint := 'True'} : "Pallet_Transport_Row_1_2";
      ST35_ST34 { S7_SetPoint := 'True'} : "Pallet_Transport_Row_1_2";
      ST33_ST34 { S7_SetPoint := 'True'} : "Pallet_Transport_Row_1_2";
      ST34_ST33 { S7_SetPoint := 'True'} : "Pallet_Transport_Row_1_2";
      ST32_ST33 { S7_SetPoint := 'True'} : "Pallet_Transport_Row_1_2";
      ST36_ST38 { S7_SetPoint := 'True'} : "Pallet_Transport_Row_1_2";
      ST38_ST36 { S7_SetPoint := 'True'} : "Pallet_Transport_Row_1_2";
      ST37_ST36 { S7_SetPoint := 'True'} : "Pallet_Transport_Row_1_2";
      ST18_ST37 { S7_SetPoint := 'True'} : "Pallet_Transport_Row_1_2";
      ST19_ST18 { S7_SetPoint := 'True'} : "Pallet_Transport_Row_1_2";
      ST20_ST19 { S7_SetPoint := 'True'} : "Pallet_Transport_Row_1_2";
      ST21_ST20 { S7_SetPoint := 'True'} : "Pallet_Transport_Row_1_2";
      ST22_ST21 { S7_SetPoint := 'True'} : "Pallet_Transport_Row_1_2";
      ST23_ST22 { S7_SetPoint := 'True'} : "Pallet_Transport_Row_1_2";
      ST24_ST23 { S7_SetPoint := 'True'} : "Pallet_Transport_Row_1_2";
      Centering_Perform : Array[7..13, 1..3] of Bool;
      Centering_Status { S7_SetPoint := 'True'} : Array[7..13, 1..3] of Bool;
      ST31_ST32 { S7_SetPoint := 'True'} : "Pallet_Transport_Row_1_2";
      ST30_ST31 { S7_SetPoint := 'True'} : "Pallet_Transport_Row_1_2";
      ST29_ST30 { S7_SetPoint := 'True'} : "Pallet_Transport_Row_1_2";
      ST28_ST29 { S7_SetPoint := 'True'} : "Pallet_Transport_Row_1_2";
      TON_Reset_Drives { S7_SetPoint := 'True'} : TON_TIME;
      TP_Reset_Drives { S7_SetPoint := 'True'} : TP_TIME;
      Reset_Drives_Var { S7_SetPoint := 'True'} : Bool;
      ST27_ST28 { S7_SetPoint := 'True'} : "Pallet_Transport_Row_1_2";
      ST26_ST27 { S7_SetPoint := 'True'} : "Pallet_Transport_Row_1_2";
      ST25_ST26 { S7_SetPoint := 'True'} : "Pallet_Transport_Row_1_2";
      tComm_W1 { S7_SetPoint := 'True'} : TON_TIME;
      tComm_W2 { S7_SetPoint := 'True'} : TON_TIME;
      tComm_W4 { S7_SetPoint := 'True'} : TON_TIME;
   END_VAR
   VAR_TEMP
      i : Int;
      Reset_Stations_Index : Int;
      Block_Check_Index : Int;
   END_VAR
BEGIN

REGION Network 1: Initialisation of pallets status
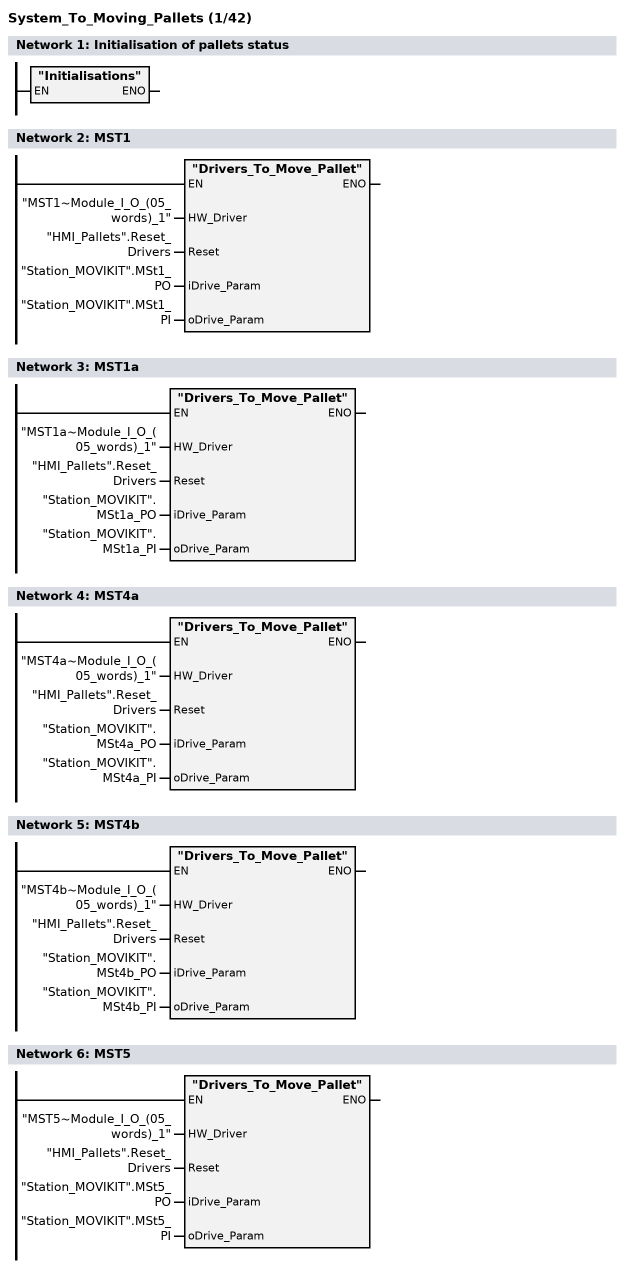
   RUNG wire#powerrail
      "Initialisations"()
   END_RUNG
   // the same network as SCL:
   "Initialisations"();
END_REGION

REGION Network 2: MST1
   RUNG wire#powerrail
      "Drivers_To_Move_Pallet"(HW_Driver := "MST1~Module_I_O_(05_words)_1", Reset := "HMI_Pallets".Reset_Drivers, iDrive_Param := "Station_MOVIKIT".MSt1_PO, oDrive_Param := "Station_MOVIKIT".MSt1_PI)
   END_RUNG
   // the same network as SCL:
   "Drivers_To_Move_Pallet"(HW_Driver := "MST1~Module_I_O_(05_words)_1",
                           Reset := "HMI_Pallets".Reset_Drivers,
                           iDrive_Param := "Station_MOVIKIT".MSt1_PO,
                           oDrive_Param := "Station_MOVIKIT".MSt1_PI);
END_REGION

REGION Network 3: MST1a
   RUNG wire#powerrail
      "Drivers_To_Move_Pallet"(HW_Driver := "MST1a~Module_I_O_(05_words)_1", Reset := "HMI_Pallets".Reset_Drivers, iDrive_Param := "Station_MOVIKIT".MSt1a_PO, oDrive_Param := "Station_MOVIKIT".MSt1a_PI)
   END_RUNG
   // the same network as SCL:
   "Drivers_To_Move_Pallet"(HW_Driver := "MST1a~Module_I_O_(05_words)_1",
                           Reset := "HMI_Pallets".Reset_Drivers,
                           iDrive_Param := "Station_MOVIKIT".MSt1a_PO,
                           oDrive_Param := "Station_MOVIKIT".MSt1a_PI);
END_REGION

REGION Network 4: MST4a
   RUNG wire#powerrail
      "Drivers_To_Move_Pallet"(HW_Driver := "MST4a~Module_I_O_(05_words)_1", Reset := "HMI_Pallets".Reset_Drivers, iDrive_Param := "Station_MOVIKIT".MSt4a_PO, oDrive_Param := "Station_MOVIKIT".MSt4a_PI)
   END_RUNG
   // the same network as SCL:
   "Drivers_To_Move_Pallet"(HW_Driver := "MST4a~Module_I_O_(05_words)_1",
                           Reset := "HMI_Pallets".Reset_Drivers,
                           iDrive_Param := "Station_MOVIKIT".MSt4a_PO,
                           oDrive_Param := "Station_MOVIKIT".MSt4a_PI);
END_REGION

REGION Network 5: MST4b
   RUNG wire#powerrail
      "Drivers_To_Move_Pallet"(HW_Driver := "MST4b~Module_I_O_(05_words)_1", Reset := "HMI_Pallets".Reset_Drivers, iDrive_Param := "Station_MOVIKIT".MSt4b_PO, oDrive_Param := "Station_MOVIKIT".MSt4b_PI)
   END_RUNG
   // the same network as SCL:
   "Drivers_To_Move_Pallet"(HW_Driver := "MST4b~Module_I_O_(05_words)_1",
                           Reset := "HMI_Pallets".Reset_Drivers,
                           iDrive_Param := "Station_MOVIKIT".MSt4b_PO,
                           oDrive_Param := "Station_MOVIKIT".MSt4b_PI);
END_REGION

REGION Network 6: MST5
   RUNG wire#powerrail
      "Drivers_To_Move_Pallet"(HW_Driver := "MST5~Module_I_O_(05_words)_1", Reset := "HMI_Pallets".Reset_Drivers, iDrive_Param := "Station_MOVIKIT".MSt5_PO, oDrive_Param := "Station_MOVIKIT".MSt5_PI)
   END_RUNG
   // the same network as SCL:
   "Drivers_To_Move_Pallet"(HW_Driver := "MST5~Module_I_O_(05_words)_1",
                           Reset := "HMI_Pallets".Reset_Drivers,
                           iDrive_Param := "Station_MOVIKIT".MSt5_PO,
                           oDrive_Param := "Station_MOVIKIT".MSt5_PI);
END_REGION

REGION Network 7: MST6a
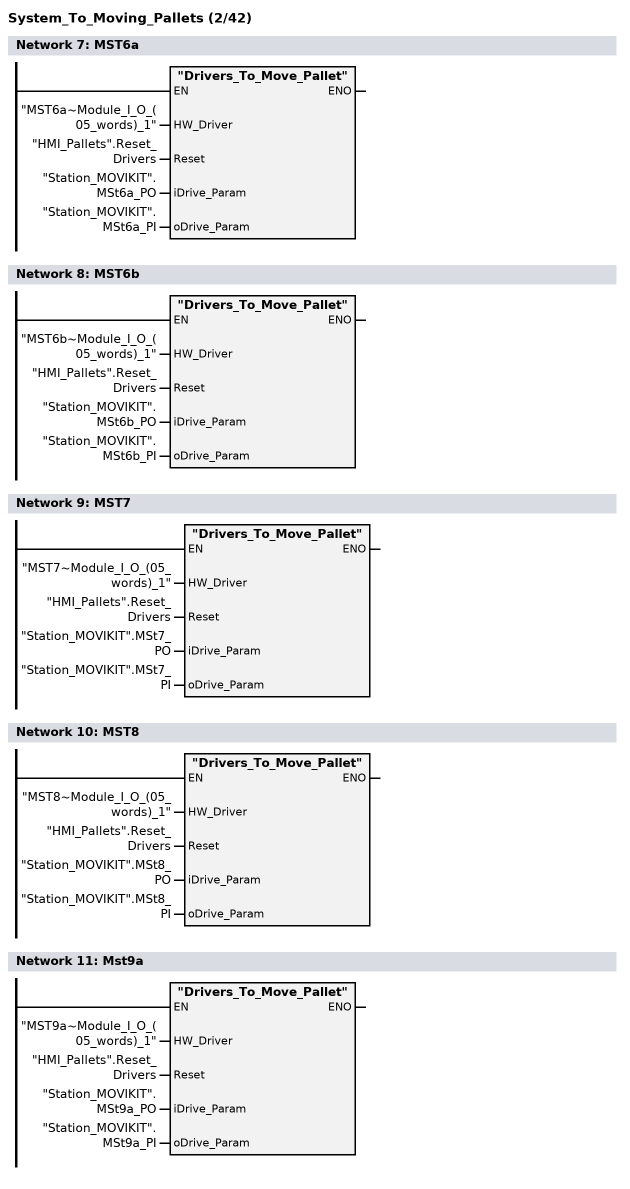
   RUNG wire#powerrail
      "Drivers_To_Move_Pallet"(HW_Driver := "MST6a~Module_I_O_(05_words)_1", Reset := "HMI_Pallets".Reset_Drivers, iDrive_Param := "Station_MOVIKIT".MSt6a_PO, oDrive_Param := "Station_MOVIKIT".MSt6a_PI)
   END_RUNG
   // the same network as SCL:
   "Drivers_To_Move_Pallet"(HW_Driver := "MST6a~Module_I_O_(05_words)_1",
                           Reset := "HMI_Pallets".Reset_Drivers,
                           iDrive_Param := "Station_MOVIKIT".MSt6a_PO,
                           oDrive_Param := "Station_MOVIKIT".MSt6a_PI);
END_REGION

REGION Network 8: MST6b
   RUNG wire#powerrail
      "Drivers_To_Move_Pallet"(HW_Driver := "MST6b~Module_I_O_(05_words)_1", Reset := "HMI_Pallets".Reset_Drivers, iDrive_Param := "Station_MOVIKIT".MSt6b_PO, oDrive_Param := "Station_MOVIKIT".MSt6b_PI)
   END_RUNG
   // the same network as SCL:
   "Drivers_To_Move_Pallet"(HW_Driver := "MST6b~Module_I_O_(05_words)_1",
                           Reset := "HMI_Pallets".Reset_Drivers,
                           iDrive_Param := "Station_MOVIKIT".MSt6b_PO,
                           oDrive_Param := "Station_MOVIKIT".MSt6b_PI);
END_REGION

REGION Network 9: MST7
   RUNG wire#powerrail
      "Drivers_To_Move_Pallet"(HW_Driver := "MST7~Module_I_O_(05_words)_1", Reset := "HMI_Pallets".Reset_Drivers, iDrive_Param := "Station_MOVIKIT".MSt7_PO, oDrive_Param := "Station_MOVIKIT".MSt7_PI)
   END_RUNG
   // the same network as SCL:
   "Drivers_To_Move_Pallet"(HW_Driver := "MST7~Module_I_O_(05_words)_1",
                           Reset := "HMI_Pallets".Reset_Drivers,
                           iDrive_Param := "Station_MOVIKIT".MSt7_PO,
                           oDrive_Param := "Station_MOVIKIT".MSt7_PI);
END_REGION

REGION Network 10: MST8
   RUNG wire#powerrail
      "Drivers_To_Move_Pallet"(HW_Driver := "MST8~Module_I_O_(05_words)_1", Reset := "HMI_Pallets".Reset_Drivers, iDrive_Param := "Station_MOVIKIT".MSt8_PO, oDrive_Param := "Station_MOVIKIT".MSt8_PI)
   END_RUNG
   // the same network as SCL:
   "Drivers_To_Move_Pallet"(HW_Driver := "MST8~Module_I_O_(05_words)_1",
                           Reset := "HMI_Pallets".Reset_Drivers,
                           iDrive_Param := "Station_MOVIKIT".MSt8_PO,
                           oDrive_Param := "Station_MOVIKIT".MSt8_PI);
END_REGION

REGION Network 11: Mst9a
   RUNG wire#powerrail
      "Drivers_To_Move_Pallet"(HW_Driver := "MST9a~Module_I_O_(05_words)_1", Reset := "HMI_Pallets".Reset_Drivers, iDrive_Param := "Station_MOVIKIT".MSt9a_PO, oDrive_Param := "Station_MOVIKIT".MSt9a_PI)
   END_RUNG
   // the same network as SCL:
   "Drivers_To_Move_Pallet"(HW_Driver := "MST9a~Module_I_O_(05_words)_1",
                           Reset := "HMI_Pallets".Reset_Drivers,
                           iDrive_Param := "Station_MOVIKIT".MSt9a_PO,
                           oDrive_Param := "Station_MOVIKIT".MSt9a_PI);
END_REGION

REGION Network 12: Mst9b
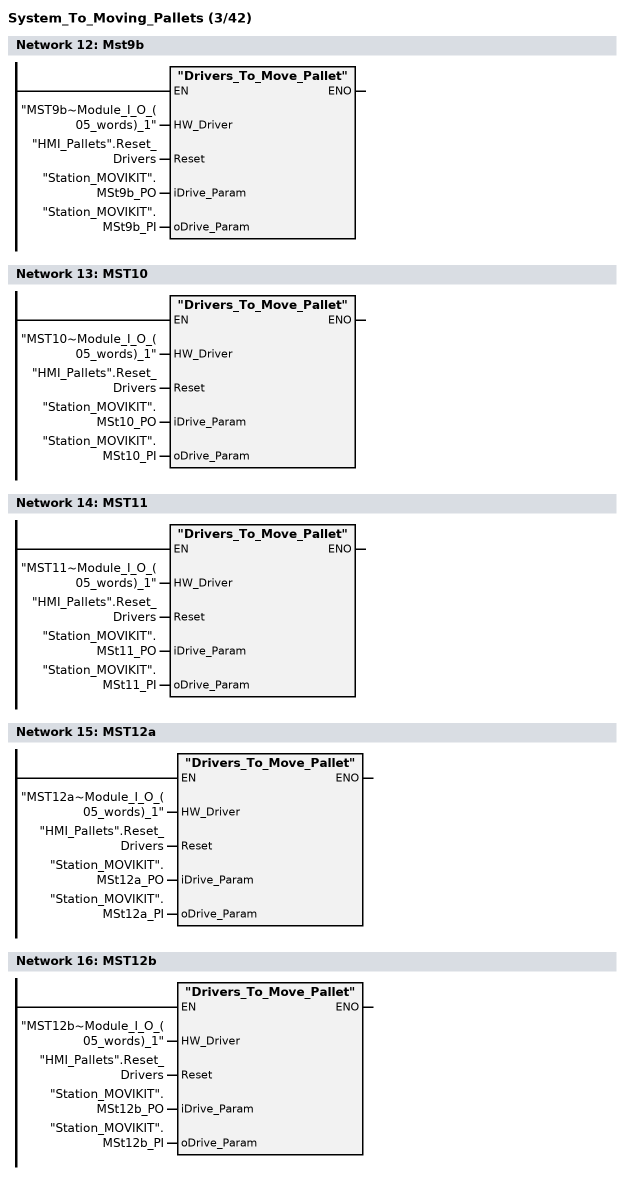
   RUNG wire#powerrail
      "Drivers_To_Move_Pallet"(HW_Driver := "MST9b~Module_I_O_(05_words)_1", Reset := "HMI_Pallets".Reset_Drivers, iDrive_Param := "Station_MOVIKIT".MSt9b_PO, oDrive_Param := "Station_MOVIKIT".MSt9b_PI)
   END_RUNG
   // the same network as SCL:
   "Drivers_To_Move_Pallet"(HW_Driver := "MST9b~Module_I_O_(05_words)_1",
                           Reset := "HMI_Pallets".Reset_Drivers,
                           iDrive_Param := "Station_MOVIKIT".MSt9b_PO,
                           oDrive_Param := "Station_MOVIKIT".MSt9b_PI);
END_REGION

REGION Network 13: MST10
   RUNG wire#powerrail
      "Drivers_To_Move_Pallet"(HW_Driver := "MST10~Module_I_O_(05_words)_1", Reset := "HMI_Pallets".Reset_Drivers, iDrive_Param := "Station_MOVIKIT".MSt10_PO, oDrive_Param := "Station_MOVIKIT".MSt10_PI)
   END_RUNG
   // the same network as SCL:
   "Drivers_To_Move_Pallet"(HW_Driver := "MST10~Module_I_O_(05_words)_1",
                           Reset := "HMI_Pallets".Reset_Drivers,
                           iDrive_Param := "Station_MOVIKIT".MSt10_PO,
                           oDrive_Param := "Station_MOVIKIT".MSt10_PI);
END_REGION

REGION Network 14: MST11
   RUNG wire#powerrail
      "Drivers_To_Move_Pallet"(HW_Driver := "MST11~Module_I_O_(05_words)_1", Reset := "HMI_Pallets".Reset_Drivers, iDrive_Param := "Station_MOVIKIT".MSt11_PO, oDrive_Param := "Station_MOVIKIT".MSt11_PI)
   END_RUNG
   // the same network as SCL:
   "Drivers_To_Move_Pallet"(HW_Driver := "MST11~Module_I_O_(05_words)_1",
                           Reset := "HMI_Pallets".Reset_Drivers,
                           iDrive_Param := "Station_MOVIKIT".MSt11_PO,
                           oDrive_Param := "Station_MOVIKIT".MSt11_PI);
END_REGION

REGION Network 15: MST12a
   RUNG wire#powerrail
      "Drivers_To_Move_Pallet"(HW_Driver := "MST12a~Module_I_O_(05_words)_1", Reset := "HMI_Pallets".Reset_Drivers, iDrive_Param := "Station_MOVIKIT".MSt12a_PO, oDrive_Param := "Station_MOVIKIT".MSt12a_PI)
   END_RUNG
   // the same network as SCL:
   "Drivers_To_Move_Pallet"(HW_Driver := "MST12a~Module_I_O_(05_words)_1",
                           Reset := "HMI_Pallets".Reset_Drivers,
                           iDrive_Param := "Station_MOVIKIT".MSt12a_PO,
                           oDrive_Param := "Station_MOVIKIT".MSt12a_PI);
END_REGION

REGION Network 16: MST12b
   RUNG wire#powerrail
      "Drivers_To_Move_Pallet"(HW_Driver := "MST12b~Module_I_O_(05_words)_1", Reset := "HMI_Pallets".Reset_Drivers, iDrive_Param := "Station_MOVIKIT".MSt12b_PO, oDrive_Param := "Station_MOVIKIT".MSt12b_PI)
   END_RUNG
   // the same network as SCL:
   "Drivers_To_Move_Pallet"(HW_Driver := "MST12b~Module_I_O_(05_words)_1",
                           Reset := "HMI_Pallets".Reset_Drivers,
                           iDrive_Param := "Station_MOVIKIT".MSt12b_PO,
                           oDrive_Param := "Station_MOVIKIT".MSt12b_PI);
END_REGION

REGION Network 17: MST13
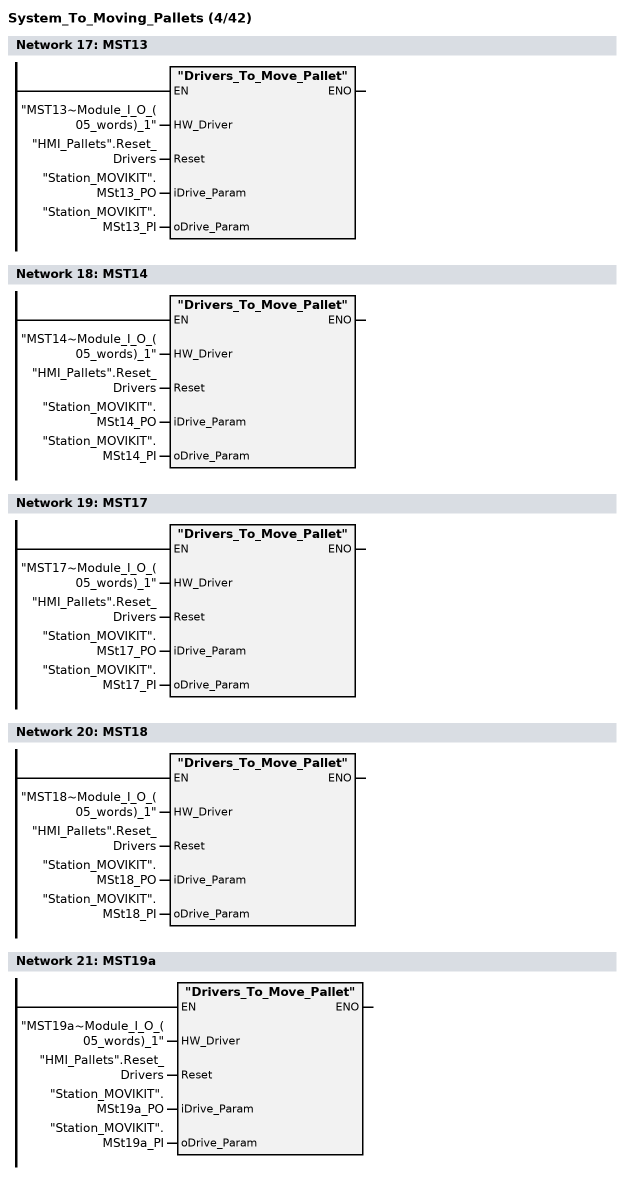
   RUNG wire#powerrail
      "Drivers_To_Move_Pallet"(HW_Driver := "MST13~Module_I_O_(05_words)_1", Reset := "HMI_Pallets".Reset_Drivers, iDrive_Param := "Station_MOVIKIT".MSt13_PO, oDrive_Param := "Station_MOVIKIT".MSt13_PI)
   END_RUNG
   // the same network as SCL:
   "Drivers_To_Move_Pallet"(HW_Driver := "MST13~Module_I_O_(05_words)_1",
                           Reset := "HMI_Pallets".Reset_Drivers,
                           iDrive_Param := "Station_MOVIKIT".MSt13_PO,
                           oDrive_Param := "Station_MOVIKIT".MSt13_PI);
END_REGION

REGION Network 18: MST14
   RUNG wire#powerrail
      "Drivers_To_Move_Pallet"(HW_Driver := "MST14~Module_I_O_(05_words)_1", Reset := "HMI_Pallets".Reset_Drivers, iDrive_Param := "Station_MOVIKIT".MSt14_PO, oDrive_Param := "Station_MOVIKIT".MSt14_PI)
   END_RUNG
   // the same network as SCL:
   "Drivers_To_Move_Pallet"(HW_Driver := "MST14~Module_I_O_(05_words)_1",
                           Reset := "HMI_Pallets".Reset_Drivers,
                           iDrive_Param := "Station_MOVIKIT".MSt14_PO,
                           oDrive_Param := "Station_MOVIKIT".MSt14_PI);
END_REGION

REGION Network 19: MST17
   RUNG wire#powerrail
      "Drivers_To_Move_Pallet"(HW_Driver := "MST17~Module_I_O_(05_words)_1", Reset := "HMI_Pallets".Reset_Drivers, iDrive_Param := "Station_MOVIKIT".MSt17_PO, oDrive_Param := "Station_MOVIKIT".MSt17_PI)
   END_RUNG
   // the same network as SCL:
   "Drivers_To_Move_Pallet"(HW_Driver := "MST17~Module_I_O_(05_words)_1",
                           Reset := "HMI_Pallets".Reset_Drivers,
                           iDrive_Param := "Station_MOVIKIT".MSt17_PO,
                           oDrive_Param := "Station_MOVIKIT".MSt17_PI);
END_REGION

REGION Network 20: MST18
   RUNG wire#powerrail
      "Drivers_To_Move_Pallet"(HW_Driver := "MST18~Module_I_O_(05_words)_1", Reset := "HMI_Pallets".Reset_Drivers, iDrive_Param := "Station_MOVIKIT".MSt18_PO, oDrive_Param := "Station_MOVIKIT".MSt18_PI)
   END_RUNG
   // the same network as SCL:
   "Drivers_To_Move_Pallet"(HW_Driver := "MST18~Module_I_O_(05_words)_1",
                           Reset := "HMI_Pallets".Reset_Drivers,
                           iDrive_Param := "Station_MOVIKIT".MSt18_PO,
                           oDrive_Param := "Station_MOVIKIT".MSt18_PI);
END_REGION

REGION Network 21: MST19a
   RUNG wire#powerrail
      "Drivers_To_Move_Pallet"(HW_Driver := "MST19a~Module_I_O_(05_words)_1", Reset := "HMI_Pallets".Reset_Drivers, iDrive_Param := "Station_MOVIKIT".MSt19a_PO, oDrive_Param := "Station_MOVIKIT".MSt19a_PI)
   END_RUNG
   // the same network as SCL:
   "Drivers_To_Move_Pallet"(HW_Driver := "MST19a~Module_I_O_(05_words)_1",
                           Reset := "HMI_Pallets".Reset_Drivers,
                           iDrive_Param := "Station_MOVIKIT".MSt19a_PO,
                           oDrive_Param := "Station_MOVIKIT".MSt19a_PI);
END_REGION

REGION Network 22: MST19b
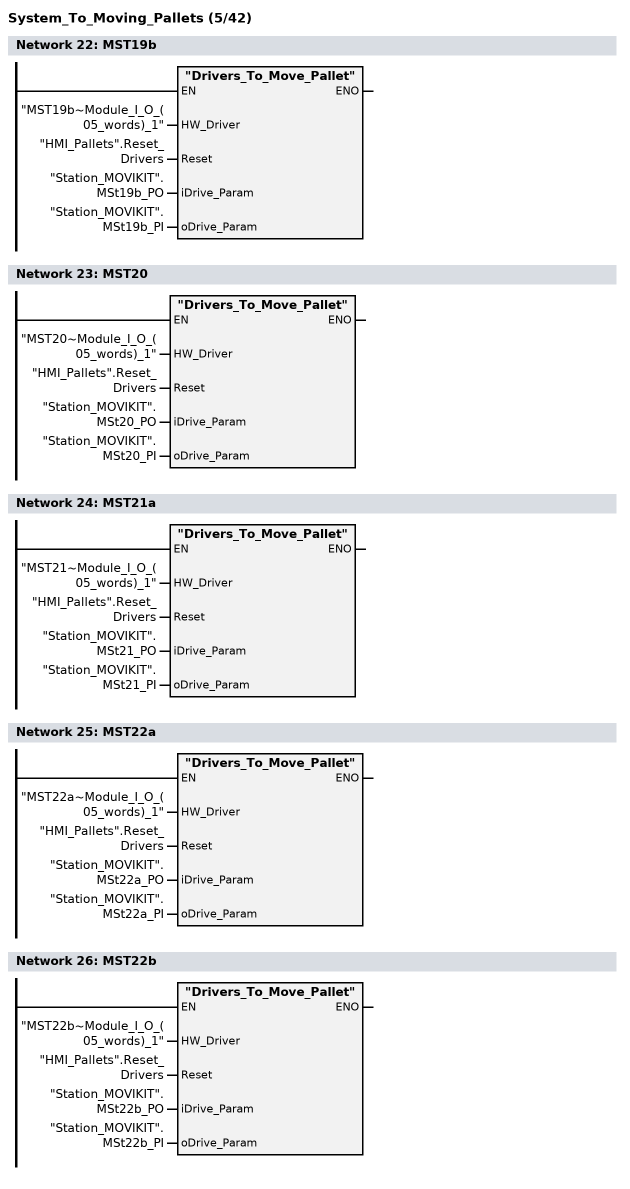
   RUNG wire#powerrail
      "Drivers_To_Move_Pallet"(HW_Driver := "MST19b~Module_I_O_(05_words)_1", Reset := "HMI_Pallets".Reset_Drivers, iDrive_Param := "Station_MOVIKIT".MSt19b_PO, oDrive_Param := "Station_MOVIKIT".MSt19b_PI)
   END_RUNG
   // the same network as SCL:
   "Drivers_To_Move_Pallet"(HW_Driver := "MST19b~Module_I_O_(05_words)_1",
                           Reset := "HMI_Pallets".Reset_Drivers,
                           iDrive_Param := "Station_MOVIKIT".MSt19b_PO,
                           oDrive_Param := "Station_MOVIKIT".MSt19b_PI);
END_REGION

REGION Network 23: MST20
   RUNG wire#powerrail
      "Drivers_To_Move_Pallet"(HW_Driver := "MST20~Module_I_O_(05_words)_1", Reset := "HMI_Pallets".Reset_Drivers, iDrive_Param := "Station_MOVIKIT".MSt20_PO, oDrive_Param := "Station_MOVIKIT".MSt20_PI)
   END_RUNG
   // the same network as SCL:
   "Drivers_To_Move_Pallet"(HW_Driver := "MST20~Module_I_O_(05_words)_1",
                           Reset := "HMI_Pallets".Reset_Drivers,
                           iDrive_Param := "Station_MOVIKIT".MSt20_PO,
                           oDrive_Param := "Station_MOVIKIT".MSt20_PI);
END_REGION

REGION Network 24: MST21a
   RUNG wire#powerrail
      "Drivers_To_Move_Pallet"(HW_Driver := "MST21~Module_I_O_(05_words)_1", Reset := "HMI_Pallets".Reset_Drivers, iDrive_Param := "Station_MOVIKIT".MSt21_PO, oDrive_Param := "Station_MOVIKIT".MSt21_PI)
   END_RUNG
   // the same network as SCL:
   "Drivers_To_Move_Pallet"(HW_Driver := "MST21~Module_I_O_(05_words)_1",
                           Reset := "HMI_Pallets".Reset_Drivers,
                           iDrive_Param := "Station_MOVIKIT".MSt21_PO,
                           oDrive_Param := "Station_MOVIKIT".MSt21_PI);
END_REGION

REGION Network 25: MST22a
   RUNG wire#powerrail
      "Drivers_To_Move_Pallet"(HW_Driver := "MST22a~Module_I_O_(05_words)_1", Reset := "HMI_Pallets".Reset_Drivers, iDrive_Param := "Station_MOVIKIT".MSt22a_PO, oDrive_Param := "Station_MOVIKIT".MSt22a_PI)
   END_RUNG
   // the same network as SCL:
   "Drivers_To_Move_Pallet"(HW_Driver := "MST22a~Module_I_O_(05_words)_1",
                           Reset := "HMI_Pallets".Reset_Drivers,
                           iDrive_Param := "Station_MOVIKIT".MSt22a_PO,
                           oDrive_Param := "Station_MOVIKIT".MSt22a_PI);
END_REGION

REGION Network 26: MST22b
   RUNG wire#powerrail
      "Drivers_To_Move_Pallet"(HW_Driver := "MST22b~Module_I_O_(05_words)_1", Reset := "HMI_Pallets".Reset_Drivers, iDrive_Param := "Station_MOVIKIT".MSt22b_PO, oDrive_Param := "Station_MOVIKIT".MSt22b_PI)
   END_RUNG
   // the same network as SCL:
   "Drivers_To_Move_Pallet"(HW_Driver := "MST22b~Module_I_O_(05_words)_1",
                           Reset := "HMI_Pallets".Reset_Drivers,
                           iDrive_Param := "Station_MOVIKIT".MSt22b_PO,
                           oDrive_Param := "Station_MOVIKIT".MSt22b_PI);
END_REGION

REGION Network 27: MST23a
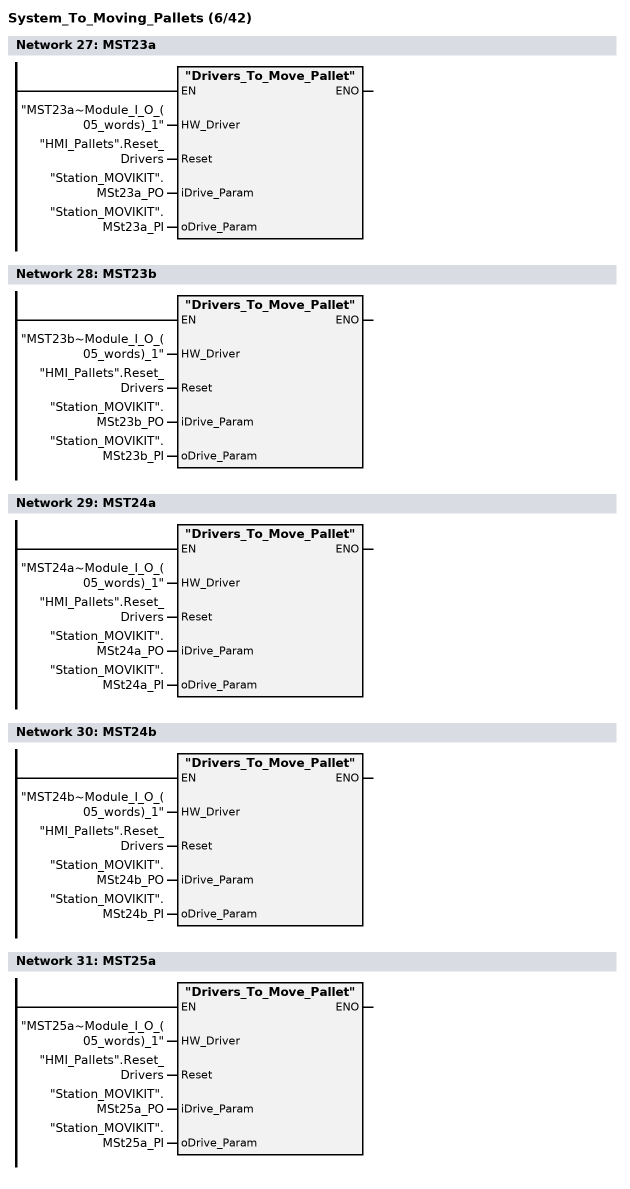
   RUNG wire#powerrail
      "Drivers_To_Move_Pallet"(HW_Driver := "MST23a~Module_I_O_(05_words)_1", Reset := "HMI_Pallets".Reset_Drivers, iDrive_Param := "Station_MOVIKIT".MSt23a_PO, oDrive_Param := "Station_MOVIKIT".MSt23a_PI)
   END_RUNG
   // the same network as SCL:
   "Drivers_To_Move_Pallet"(HW_Driver := "MST23a~Module_I_O_(05_words)_1",
                           Reset := "HMI_Pallets".Reset_Drivers,
                           iDrive_Param := "Station_MOVIKIT".MSt23a_PO,
                           oDrive_Param := "Station_MOVIKIT".MSt23a_PI);
END_REGION

REGION Network 28: MST23b
   RUNG wire#powerrail
      "Drivers_To_Move_Pallet"(HW_Driver := "MST23b~Module_I_O_(05_words)_1", Reset := "HMI_Pallets".Reset_Drivers, iDrive_Param := "Station_MOVIKIT".MSt23b_PO, oDrive_Param := "Station_MOVIKIT".MSt23b_PI)
   END_RUNG
   // the same network as SCL:
   "Drivers_To_Move_Pallet"(HW_Driver := "MST23b~Module_I_O_(05_words)_1",
                           Reset := "HMI_Pallets".Reset_Drivers,
                           iDrive_Param := "Station_MOVIKIT".MSt23b_PO,
                           oDrive_Param := "Station_MOVIKIT".MSt23b_PI);
END_REGION

REGION Network 29: MST24a
   RUNG wire#powerrail
      "Drivers_To_Move_Pallet"(HW_Driver := "MST24a~Module_I_O_(05_words)_1", Reset := "HMI_Pallets".Reset_Drivers, iDrive_Param := "Station_MOVIKIT".MSt24a_PO, oDrive_Param := "Station_MOVIKIT".MSt24a_PI)
   END_RUNG
   // the same network as SCL:
   "Drivers_To_Move_Pallet"(HW_Driver := "MST24a~Module_I_O_(05_words)_1",
                           Reset := "HMI_Pallets".Reset_Drivers,
                           iDrive_Param := "Station_MOVIKIT".MSt24a_PO,
                           oDrive_Param := "Station_MOVIKIT".MSt24a_PI);
END_REGION

REGION Network 30: MST24b
   RUNG wire#powerrail
      "Drivers_To_Move_Pallet"(HW_Driver := "MST24b~Module_I_O_(05_words)_1", Reset := "HMI_Pallets".Reset_Drivers, iDrive_Param := "Station_MOVIKIT".MSt24b_PO, oDrive_Param := "Station_MOVIKIT".MSt24b_PI)
   END_RUNG
   // the same network as SCL:
   "Drivers_To_Move_Pallet"(HW_Driver := "MST24b~Module_I_O_(05_words)_1",
                           Reset := "HMI_Pallets".Reset_Drivers,
                           iDrive_Param := "Station_MOVIKIT".MSt24b_PO,
                           oDrive_Param := "Station_MOVIKIT".MSt24b_PI);
END_REGION

REGION Network 31: MST25a
   RUNG wire#powerrail
      "Drivers_To_Move_Pallet"(HW_Driver := "MST25a~Module_I_O_(05_words)_1", Reset := "HMI_Pallets".Reset_Drivers, iDrive_Param := "Station_MOVIKIT".MSt25a_PO, oDrive_Param := "Station_MOVIKIT".MSt25a_PI)
   END_RUNG
   // the same network as SCL:
   "Drivers_To_Move_Pallet"(HW_Driver := "MST25a~Module_I_O_(05_words)_1",
                           Reset := "HMI_Pallets".Reset_Drivers,
                           iDrive_Param := "Station_MOVIKIT".MSt25a_PO,
                           oDrive_Param := "Station_MOVIKIT".MSt25a_PI);
END_REGION

REGION Network 32: MST25b
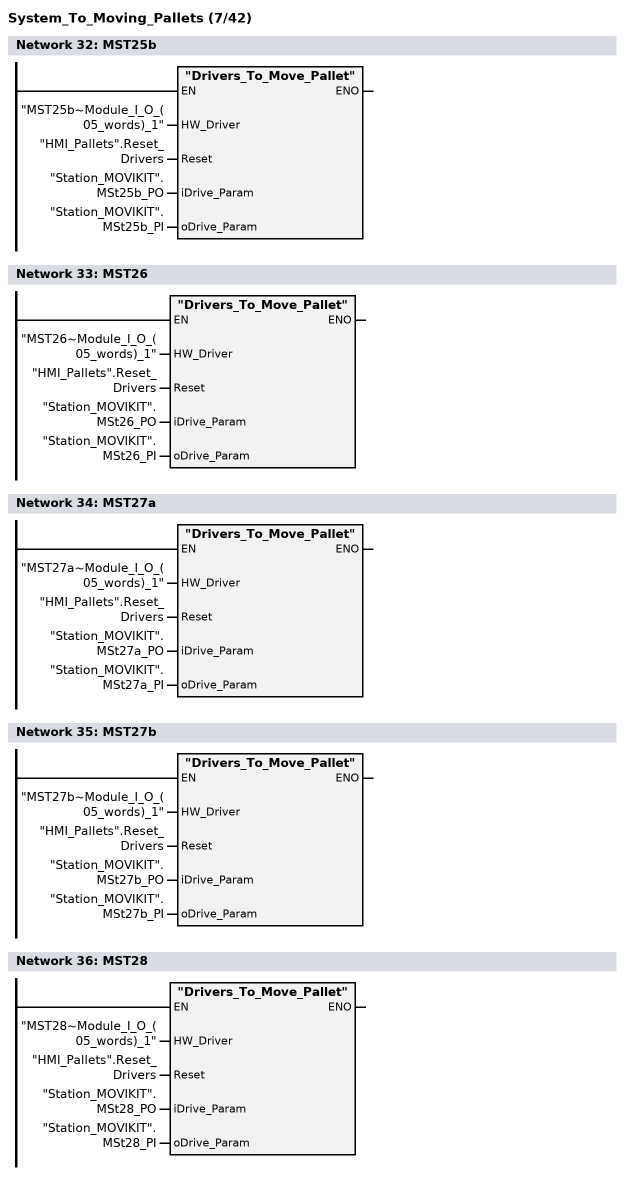
   RUNG wire#powerrail
      "Drivers_To_Move_Pallet"(HW_Driver := "MST25b~Module_I_O_(05_words)_1", Reset := "HMI_Pallets".Reset_Drivers, iDrive_Param := "Station_MOVIKIT".MSt25b_PO, oDrive_Param := "Station_MOVIKIT".MSt25b_PI)
   END_RUNG
   // the same network as SCL:
   "Drivers_To_Move_Pallet"(HW_Driver := "MST25b~Module_I_O_(05_words)_1",
                           Reset := "HMI_Pallets".Reset_Drivers,
                           iDrive_Param := "Station_MOVIKIT".MSt25b_PO,
                           oDrive_Param := "Station_MOVIKIT".MSt25b_PI);
END_REGION

REGION Network 33: MST26
   RUNG wire#powerrail
      "Drivers_To_Move_Pallet"(HW_Driver := "MST26~Module_I_O_(05_words)_1", Reset := "HMI_Pallets".Reset_Drivers, iDrive_Param := "Station_MOVIKIT".MSt26_PO, oDrive_Param := "Station_MOVIKIT".MSt26_PI)
   END_RUNG
   // the same network as SCL:
   "Drivers_To_Move_Pallet"(HW_Driver := "MST26~Module_I_O_(05_words)_1",
                           Reset := "HMI_Pallets".Reset_Drivers,
                           iDrive_Param := "Station_MOVIKIT".MSt26_PO,
                           oDrive_Param := "Station_MOVIKIT".MSt26_PI);
END_REGION

REGION Network 34: MST27a
   RUNG wire#powerrail
      "Drivers_To_Move_Pallet"(HW_Driver := "MST27a~Module_I_O_(05_words)_1", Reset := "HMI_Pallets".Reset_Drivers, iDrive_Param := "Station_MOVIKIT".MSt27a_PO, oDrive_Param := "Station_MOVIKIT".MSt27a_PI)
   END_RUNG
   // the same network as SCL:
   "Drivers_To_Move_Pallet"(HW_Driver := "MST27a~Module_I_O_(05_words)_1",
                           Reset := "HMI_Pallets".Reset_Drivers,
                           iDrive_Param := "Station_MOVIKIT".MSt27a_PO,
                           oDrive_Param := "Station_MOVIKIT".MSt27a_PI);
END_REGION

REGION Network 35: MST27b
   RUNG wire#powerrail
      "Drivers_To_Move_Pallet"(HW_Driver := "MST27b~Module_I_O_(05_words)_1", Reset := "HMI_Pallets".Reset_Drivers, iDrive_Param := "Station_MOVIKIT".MSt27b_PO, oDrive_Param := "Station_MOVIKIT".MSt27b_PI)
   END_RUNG
   // the same network as SCL:
   "Drivers_To_Move_Pallet"(HW_Driver := "MST27b~Module_I_O_(05_words)_1",
                           Reset := "HMI_Pallets".Reset_Drivers,
                           iDrive_Param := "Station_MOVIKIT".MSt27b_PO,
                           oDrive_Param := "Station_MOVIKIT".MSt27b_PI);
END_REGION

REGION Network 36: MST28
   RUNG wire#powerrail
      "Drivers_To_Move_Pallet"(HW_Driver := "MST28~Module_I_O_(05_words)_1", Reset := "HMI_Pallets".Reset_Drivers, iDrive_Param := "Station_MOVIKIT".MSt28_PO, oDrive_Param := "Station_MOVIKIT".MSt28_PI)
   END_RUNG
   // the same network as SCL:
   "Drivers_To_Move_Pallet"(HW_Driver := "MST28~Module_I_O_(05_words)_1",
                           Reset := "HMI_Pallets".Reset_Drivers,
                           iDrive_Param := "Station_MOVIKIT".MSt28_PO,
                           oDrive_Param := "Station_MOVIKIT".MSt28_PI);
END_REGION

REGION Network 37: MST29
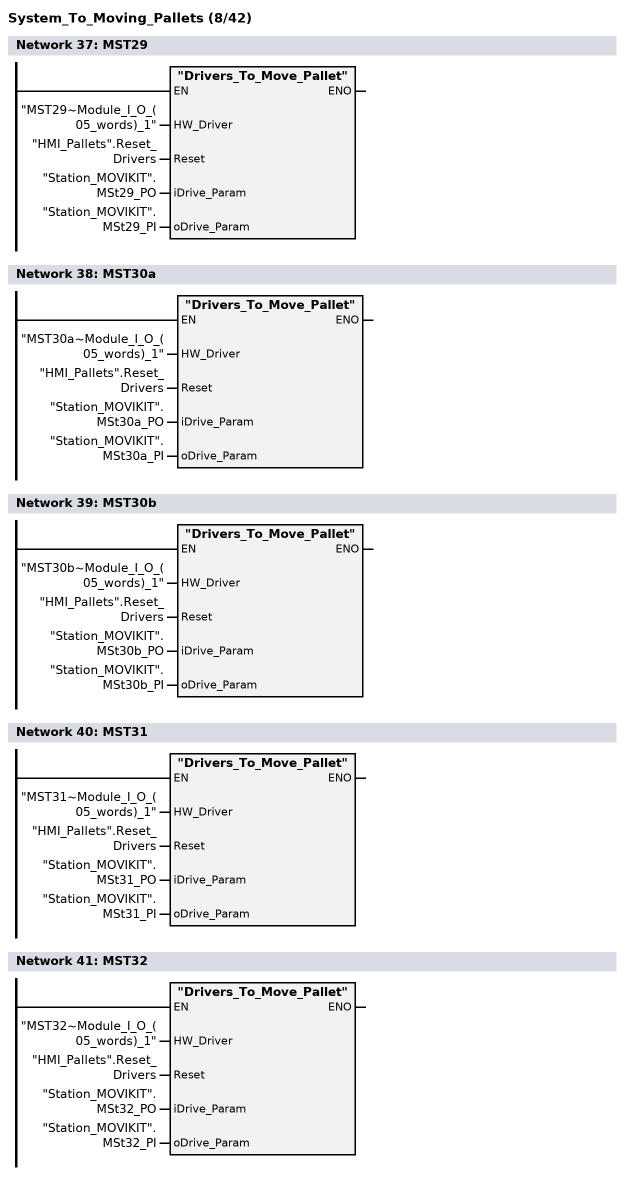
   RUNG wire#powerrail
      "Drivers_To_Move_Pallet"(HW_Driver := "MST29~Module_I_O_(05_words)_1", Reset := "HMI_Pallets".Reset_Drivers, iDrive_Param := "Station_MOVIKIT".MSt29_PO, oDrive_Param := "Station_MOVIKIT".MSt29_PI)
   END_RUNG
   // the same network as SCL:
   "Drivers_To_Move_Pallet"(HW_Driver := "MST29~Module_I_O_(05_words)_1",
                           Reset := "HMI_Pallets".Reset_Drivers,
                           iDrive_Param := "Station_MOVIKIT".MSt29_PO,
                           oDrive_Param := "Station_MOVIKIT".MSt29_PI);
END_REGION

REGION Network 38: MST30a
   RUNG wire#powerrail
      "Drivers_To_Move_Pallet"(HW_Driver := "MST30a~Module_I_O_(05_words)_1", Reset := "HMI_Pallets".Reset_Drivers, iDrive_Param := "Station_MOVIKIT".MSt30a_PO, oDrive_Param := "Station_MOVIKIT".MSt30a_PI)
   END_RUNG
   // the same network as SCL:
   "Drivers_To_Move_Pallet"(HW_Driver := "MST30a~Module_I_O_(05_words)_1",
                           Reset := "HMI_Pallets".Reset_Drivers,
                           iDrive_Param := "Station_MOVIKIT".MSt30a_PO,
                           oDrive_Param := "Station_MOVIKIT".MSt30a_PI);
END_REGION

REGION Network 39: MST30b
   RUNG wire#powerrail
      "Drivers_To_Move_Pallet"(HW_Driver := "MST30b~Module_I_O_(05_words)_1", Reset := "HMI_Pallets".Reset_Drivers, iDrive_Param := "Station_MOVIKIT".MSt30b_PO, oDrive_Param := "Station_MOVIKIT".MSt30b_PI)
   END_RUNG
   // the same network as SCL:
   "Drivers_To_Move_Pallet"(HW_Driver := "MST30b~Module_I_O_(05_words)_1",
                           Reset := "HMI_Pallets".Reset_Drivers,
                           iDrive_Param := "Station_MOVIKIT".MSt30b_PO,
                           oDrive_Param := "Station_MOVIKIT".MSt30b_PI);
END_REGION

REGION Network 40: MST31
   RUNG wire#powerrail
      "Drivers_To_Move_Pallet"(HW_Driver := "MST31~Module_I_O_(05_words)_1", Reset := "HMI_Pallets".Reset_Drivers, iDrive_Param := "Station_MOVIKIT".MSt31_PO, oDrive_Param := "Station_MOVIKIT".MSt31_PI)
   END_RUNG
   // the same network as SCL:
   "Drivers_To_Move_Pallet"(HW_Driver := "MST31~Module_I_O_(05_words)_1",
                           Reset := "HMI_Pallets".Reset_Drivers,
                           iDrive_Param := "Station_MOVIKIT".MSt31_PO,
                           oDrive_Param := "Station_MOVIKIT".MSt31_PI);
END_REGION

REGION Network 41: MST32
   RUNG wire#powerrail
      "Drivers_To_Move_Pallet"(HW_Driver := "MST32~Module_I_O_(05_words)_1", Reset := "HMI_Pallets".Reset_Drivers, iDrive_Param := "Station_MOVIKIT".MSt32_PO, oDrive_Param := "Station_MOVIKIT".MSt32_PI)
   END_RUNG
   // the same network as SCL:
   "Drivers_To_Move_Pallet"(HW_Driver := "MST32~Module_I_O_(05_words)_1",
                           Reset := "HMI_Pallets".Reset_Drivers,
                           iDrive_Param := "Station_MOVIKIT".MSt32_PO,
                           oDrive_Param := "Station_MOVIKIT".MSt32_PI);
END_REGION

REGION Network 42: MST33a
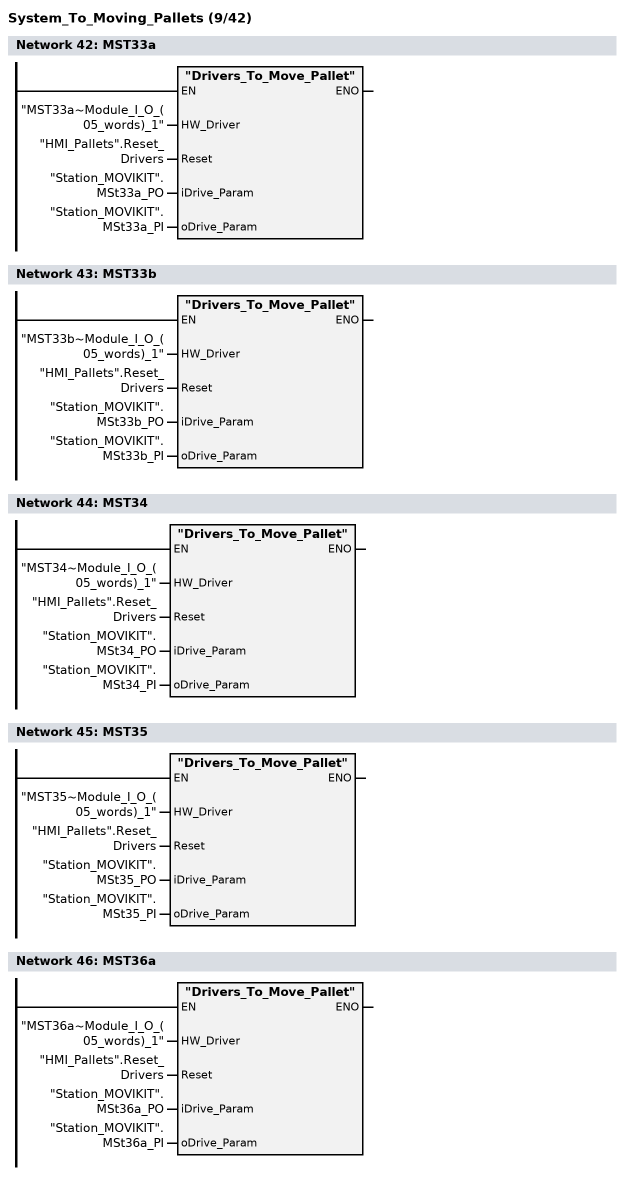
   RUNG wire#powerrail
      "Drivers_To_Move_Pallet"(HW_Driver := "MST33a~Module_I_O_(05_words)_1", Reset := "HMI_Pallets".Reset_Drivers, iDrive_Param := "Station_MOVIKIT".MSt33a_PO, oDrive_Param := "Station_MOVIKIT".MSt33a_PI)
   END_RUNG
   // the same network as SCL:
   "Drivers_To_Move_Pallet"(HW_Driver := "MST33a~Module_I_O_(05_words)_1",
                           Reset := "HMI_Pallets".Reset_Drivers,
                           iDrive_Param := "Station_MOVIKIT".MSt33a_PO,
                           oDrive_Param := "Station_MOVIKIT".MSt33a_PI);
END_REGION

REGION Network 43: MST33b
   RUNG wire#powerrail
      "Drivers_To_Move_Pallet"(HW_Driver := "MST33b~Module_I_O_(05_words)_1", Reset := "HMI_Pallets".Reset_Drivers, iDrive_Param := "Station_MOVIKIT".MSt33b_PO, oDrive_Param := "Station_MOVIKIT".MSt33b_PI)
   END_RUNG
   // the same network as SCL:
   "Drivers_To_Move_Pallet"(HW_Driver := "MST33b~Module_I_O_(05_words)_1",
                           Reset := "HMI_Pallets".Reset_Drivers,
                           iDrive_Param := "Station_MOVIKIT".MSt33b_PO,
                           oDrive_Param := "Station_MOVIKIT".MSt33b_PI);
END_REGION

REGION Network 44: MST34
   RUNG wire#powerrail
      "Drivers_To_Move_Pallet"(HW_Driver := "MST34~Module_I_O_(05_words)_1", Reset := "HMI_Pallets".Reset_Drivers, iDrive_Param := "Station_MOVIKIT".MSt34_PO, oDrive_Param := "Station_MOVIKIT".MSt34_PI)
   END_RUNG
   // the same network as SCL:
   "Drivers_To_Move_Pallet"(HW_Driver := "MST34~Module_I_O_(05_words)_1",
                           Reset := "HMI_Pallets".Reset_Drivers,
                           iDrive_Param := "Station_MOVIKIT".MSt34_PO,
                           oDrive_Param := "Station_MOVIKIT".MSt34_PI);
END_REGION

REGION Network 45: MST35
   RUNG wire#powerrail
      "Drivers_To_Move_Pallet"(HW_Driver := "MST35~Module_I_O_(05_words)_1", Reset := "HMI_Pallets".Reset_Drivers, iDrive_Param := "Station_MOVIKIT".MSt35_PO, oDrive_Param := "Station_MOVIKIT".MSt35_PI)
   END_RUNG
   // the same network as SCL:
   "Drivers_To_Move_Pallet"(HW_Driver := "MST35~Module_I_O_(05_words)_1",
                           Reset := "HMI_Pallets".Reset_Drivers,
                           iDrive_Param := "Station_MOVIKIT".MSt35_PO,
                           oDrive_Param := "Station_MOVIKIT".MSt35_PI);
END_REGION

REGION Network 46: MST36a
   RUNG wire#powerrail
      "Drivers_To_Move_Pallet"(HW_Driver := "MST36a~Module_I_O_(05_words)_1", Reset := "HMI_Pallets".Reset_Drivers, iDrive_Param := "Station_MOVIKIT".MSt36a_PO, oDrive_Param := "Station_MOVIKIT".MSt36a_PI)
   END_RUNG
   // the same network as SCL:
   "Drivers_To_Move_Pallet"(HW_Driver := "MST36a~Module_I_O_(05_words)_1",
                           Reset := "HMI_Pallets".Reset_Drivers,
                           iDrive_Param := "Station_MOVIKIT".MSt36a_PO,
                           oDrive_Param := "Station_MOVIKIT".MSt36a_PI);
END_REGION

REGION Network 47: MST36b
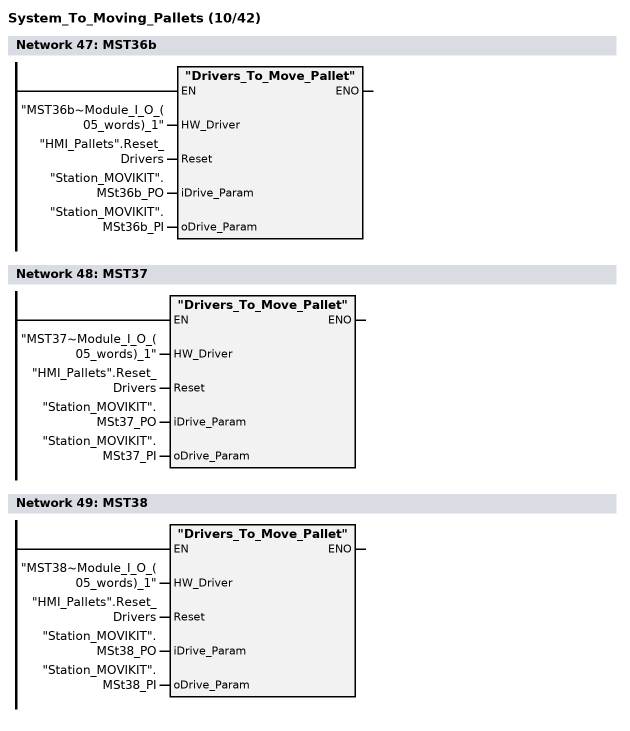
   RUNG wire#powerrail
      "Drivers_To_Move_Pallet"(HW_Driver := "MST36b~Module_I_O_(05_words)_1", Reset := "HMI_Pallets".Reset_Drivers, iDrive_Param := "Station_MOVIKIT".MSt36b_PO, oDrive_Param := "Station_MOVIKIT".MSt36b_PI)
   END_RUNG
   // the same network as SCL:
   "Drivers_To_Move_Pallet"(HW_Driver := "MST36b~Module_I_O_(05_words)_1",
                           Reset := "HMI_Pallets".Reset_Drivers,
                           iDrive_Param := "Station_MOVIKIT".MSt36b_PO,
                           oDrive_Param := "Station_MOVIKIT".MSt36b_PI);
END_REGION

REGION Network 48: MST37
   RUNG wire#powerrail
      "Drivers_To_Move_Pallet"(HW_Driver := "MST37~Module_I_O_(05_words)_1", Reset := "HMI_Pallets".Reset_Drivers, iDrive_Param := "Station_MOVIKIT".MSt37_PO, oDrive_Param := "Station_MOVIKIT".MSt37_PI)
   END_RUNG
   // the same network as SCL:
   "Drivers_To_Move_Pallet"(HW_Driver := "MST37~Module_I_O_(05_words)_1",
                           Reset := "HMI_Pallets".Reset_Drivers,
                           iDrive_Param := "Station_MOVIKIT".MSt37_PO,
                           oDrive_Param := "Station_MOVIKIT".MSt37_PI);
END_REGION

REGION Network 49: MST38
   RUNG wire#powerrail
      "Drivers_To_Move_Pallet"(HW_Driver := "MST38~Module_I_O_(05_words)_1", Reset := "HMI_Pallets".Reset_Drivers, iDrive_Param := "Station_MOVIKIT".MSt38_PO, oDrive_Param := "Station_MOVIKIT".MSt38_PI)
   END_RUNG
   // the same network as SCL:
   "Drivers_To_Move_Pallet"(HW_Driver := "MST38~Module_I_O_(05_words)_1",
                           Reset := "HMI_Pallets".Reset_Drivers,
                           iDrive_Param := "Station_MOVIKIT".MSt38_PO,
                           oDrive_Param := "Station_MOVIKIT".MSt38_PI);
END_REGION

REGION Network 50 (SCL): Clean Movment
   "Clean_Movment"(Arr := "HMI_Pallets".Run_Command_left_ROW1);
   "Clean_Movment"(Arr := "HMI_Pallets".Run_Command_left_ROW2);
   "Clean_Movment"(Arr := "HMI_Pallets".Run_Command_left_ROW3);
   "Clean_Movment"(Arr := "HMI_Pallets".Run_Command_left_ROW4);

   "Clean_Movment"(Arr := "HMI_Pallets".Run_Command_right_ROW1);
   "Clean_Movment"(Arr := "HMI_Pallets".Run_Command_right_ROW2);
   "Clean_Movment"(Arr := "HMI_Pallets".Run_Command_right_ROW3);
   "Clean_Movment"(Arr := "HMI_Pallets".Run_Command_right_ROW4);
END_REGION

REGION Network 51: ST13->ST14
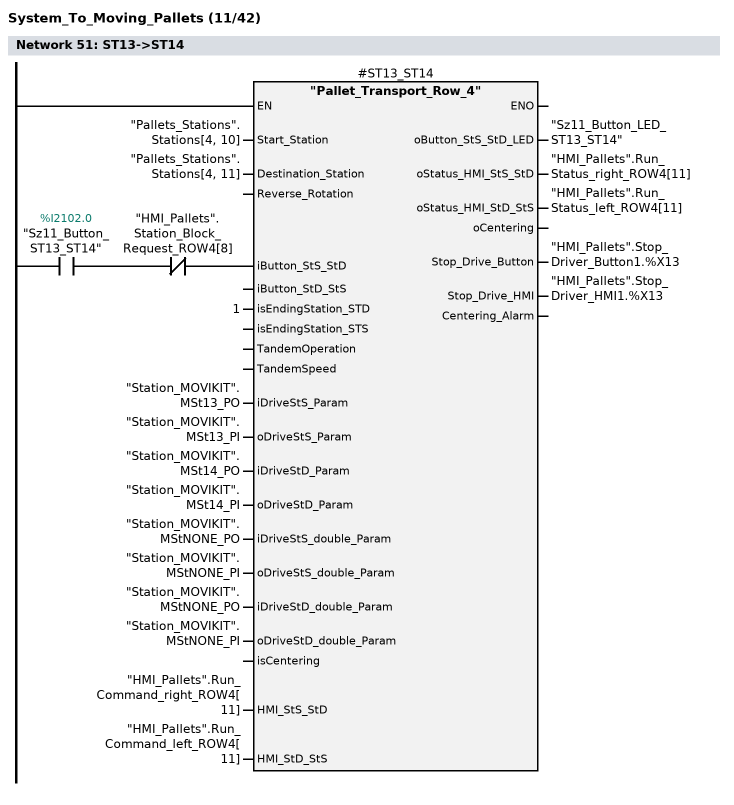
   RUNG wire#powerrail
      #ST13_ST14(iButton_StS_StD := wire#w1, Start_Station := "Pallets_Stations".Stations[4, 10], Destination_Station := "Pallets_Stations".Stations[4, 11], Reverse_Rotation :=, iButton_StD_StS :=, isEndingStation_STD := 1, isEndingStation_STS :=, TandemOperation :=, TandemSpeed :=, iDriveStS_Param := "Station_MOVIKIT".MSt13_PO, oDriveStS_Param := "Station_MOVIKIT".MSt13_PI, iDriveStD_Param := "Station_MOVIKIT".MSt14_PO, oDriveStD_Param := "Station_MOVIKIT".MSt14_PI, iDriveStS_double_Param := "Station_MOVIKIT".MStNONE_PO, oDriveStS_double_Param := "Station_MOVIKIT".MStNONE_PI, iDriveStD_double_Param := "Station_MOVIKIT".MStNONE_PO, oDriveStD_double_Param := "Station_MOVIKIT".MStNONE_PI, isCentering :=, HMI_StS_StD := "HMI_Pallets".Run_Command_right_ROW4[11], HMI_StD_StS := "HMI_Pallets".Run_Command_left_ROW4[11], oButton_StS_StD_LED => "Sz11_Button_LED_ST13_ST14", oStatus_HMI_StS_StD => "HMI_Pallets".Run_Status_right_ROW4[11], oStatus_HMI_StD_StS => "HMI_Pallets".Run_Status_left_ROW4[11], oCentering =>, Stop_Drive_Button => "HMI_Pallets".Stop_Driver_Button1.%X13, Stop_Drive_HMI => "HMI_Pallets".Stop_Driver_HMI1.%X13, Centering_Alarm =>)
   END_RUNG
   RUNG wire#powerrail
      Contact( "Sz11_Button_ST13_ST14" )
      I_Contact( "HMI_Pallets".Station_Block_Request_ROW4[8] )
   END_RUNG wire#w1
   // the same network as SCL:
   #ST13_ST14(Start_Station := "Pallets_Stations".Stations[4, 10],   // "Pallet_Transport_Row_4"
              Destination_Station := "Pallets_Stations".Stations[4, 11],
              iButton_StS_StD := "Sz11_Button_ST13_ST14" AND NOT "HMI_Pallets".Station_Block_Request_ROW4[8],
              isEndingStation_STD := 1,
              iDriveStS_Param := "Station_MOVIKIT".MSt13_PO,
              oDriveStS_Param := "Station_MOVIKIT".MSt13_PI,
              iDriveStD_Param := "Station_MOVIKIT".MSt14_PO,
              oDriveStD_Param := "Station_MOVIKIT".MSt14_PI,
              iDriveStS_double_Param := "Station_MOVIKIT".MStNONE_PO,
              oDriveStS_double_Param := "Station_MOVIKIT".MStNONE_PI,
              iDriveStD_double_Param := "Station_MOVIKIT".MStNONE_PO,
              oDriveStD_double_Param := "Station_MOVIKIT".MStNONE_PI,
              HMI_StS_StD := "HMI_Pallets".Run_Command_right_ROW4[11],
              HMI_StD_StS := "HMI_Pallets".Run_Command_left_ROW4[11],
              oButton_StS_StD_LED => "Sz11_Button_LED_ST13_ST14",
              oStatus_HMI_StS_StD => "HMI_Pallets".Run_Status_right_ROW4[11],
              oStatus_HMI_StD_StS => "HMI_Pallets".Run_Status_left_ROW4[11],
              Stop_Drive_Button => "HMI_Pallets".Stop_Driver_Button1.%X13,
              Stop_Drive_HMI => "HMI_Pallets".Stop_Driver_HMI1.%X13);
END_REGION

REGION Network 52: ST12->ST13
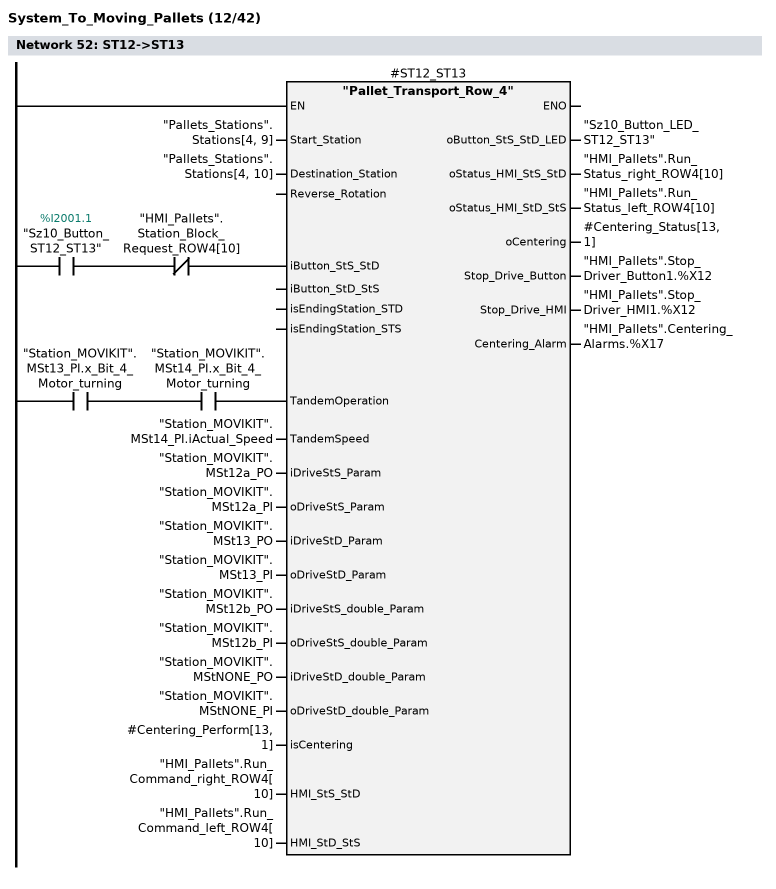
   RUNG wire#powerrail
      #ST12_ST13(iButton_StS_StD := wire#w1, TandemOperation := wire#w2, Start_Station := "Pallets_Stations".Stations[4, 9], Destination_Station := "Pallets_Stations".Stations[4, 10], Reverse_Rotation :=, iButton_StD_StS :=, isEndingStation_STD :=, isEndingStation_STS :=, TandemSpeed := "Station_MOVIKIT".MSt14_PI.iActual_Speed, iDriveStS_Param := "Station_MOVIKIT".MSt12a_PO, oDriveStS_Param := "Station_MOVIKIT".MSt12a_PI, iDriveStD_Param := "Station_MOVIKIT".MSt13_PO, oDriveStD_Param := "Station_MOVIKIT".MSt13_PI, iDriveStS_double_Param := "Station_MOVIKIT".MSt12b_PO, oDriveStS_double_Param := "Station_MOVIKIT".MSt12b_PI, iDriveStD_double_Param := "Station_MOVIKIT".MStNONE_PO, oDriveStD_double_Param := "Station_MOVIKIT".MStNONE_PI, isCentering := #Centering_Perform[13, 1], HMI_StS_StD := "HMI_Pallets".Run_Command_right_ROW4[10], HMI_StD_StS := "HMI_Pallets".Run_Command_left_ROW4[10], oButton_StS_StD_LED => "Sz10_Button_LED_ST12_ST13", oStatus_HMI_StS_StD => "HMI_Pallets".Run_Status_right_ROW4[10], oStatus_HMI_StD_StS => "HMI_Pallets".Run_Status_left_ROW4[10], oCentering => #Centering_Status[13, 1], Stop_Drive_Button => "HMI_Pallets".Stop_Driver_Button1.%X12, Stop_Drive_HMI => "HMI_Pallets".Stop_Driver_HMI1.%X12, Centering_Alarm => "HMI_Pallets".Centering_Alarms.%X17)
   END_RUNG
   RUNG wire#powerrail
      Contact( "Sz10_Button_ST12_ST13" )
      I_Contact( "HMI_Pallets".Station_Block_Request_ROW4[10] )
   END_RUNG wire#w1
   RUNG wire#powerrail
      Contact( "Station_MOVIKIT".MSt13_PI.x_Bit_4_Motor_turning )
      Contact( "Station_MOVIKIT".MSt14_PI.x_Bit_4_Motor_turning )
   END_RUNG wire#w2
   // the same network as SCL:
   #ST12_ST13(Start_Station := "Pallets_Stations".Stations[4, 9],   // "Pallet_Transport_Row_4"
              Destination_Station := "Pallets_Stations".Stations[4, 10],
              iButton_StS_StD := "Sz10_Button_ST12_ST13" AND NOT "HMI_Pallets".Station_Block_Request_ROW4[10],
              TandemOperation := "Station_MOVIKIT".MSt13_PI.x_Bit_4_Motor_turning AND "Station_MOVIKIT".MSt14_PI.x_Bit_4_Motor_turning,
              TandemSpeed := "Station_MOVIKIT".MSt14_PI.iActual_Speed,
              iDriveStS_Param := "Station_MOVIKIT".MSt12a_PO,
              oDriveStS_Param := "Station_MOVIKIT".MSt12a_PI,
              iDriveStD_Param := "Station_MOVIKIT".MSt13_PO,
              oDriveStD_Param := "Station_MOVIKIT".MSt13_PI,
              iDriveStS_double_Param := "Station_MOVIKIT".MSt12b_PO,
              oDriveStS_double_Param := "Station_MOVIKIT".MSt12b_PI,
              iDriveStD_double_Param := "Station_MOVIKIT".MStNONE_PO,
              oDriveStD_double_Param := "Station_MOVIKIT".MStNONE_PI,
              isCentering := #Centering_Perform[13, 1],
              HMI_StS_StD := "HMI_Pallets".Run_Command_right_ROW4[10],
              HMI_StD_StS := "HMI_Pallets".Run_Command_left_ROW4[10],
              oButton_StS_StD_LED => "Sz10_Button_LED_ST12_ST13",
              oStatus_HMI_StS_StD => "HMI_Pallets".Run_Status_right_ROW4[10],
              oStatus_HMI_StD_StS => "HMI_Pallets".Run_Status_left_ROW4[10],
              oCentering => #Centering_Status[13, 1],
              Stop_Drive_Button => "HMI_Pallets".Stop_Driver_Button1.%X12,
              Stop_Drive_HMI => "HMI_Pallets".Stop_Driver_HMI1.%X12,
              Centering_Alarm => "HMI_Pallets".Centering_Alarms.%X17);
END_REGION

REGION Network 53: ST11->ST12
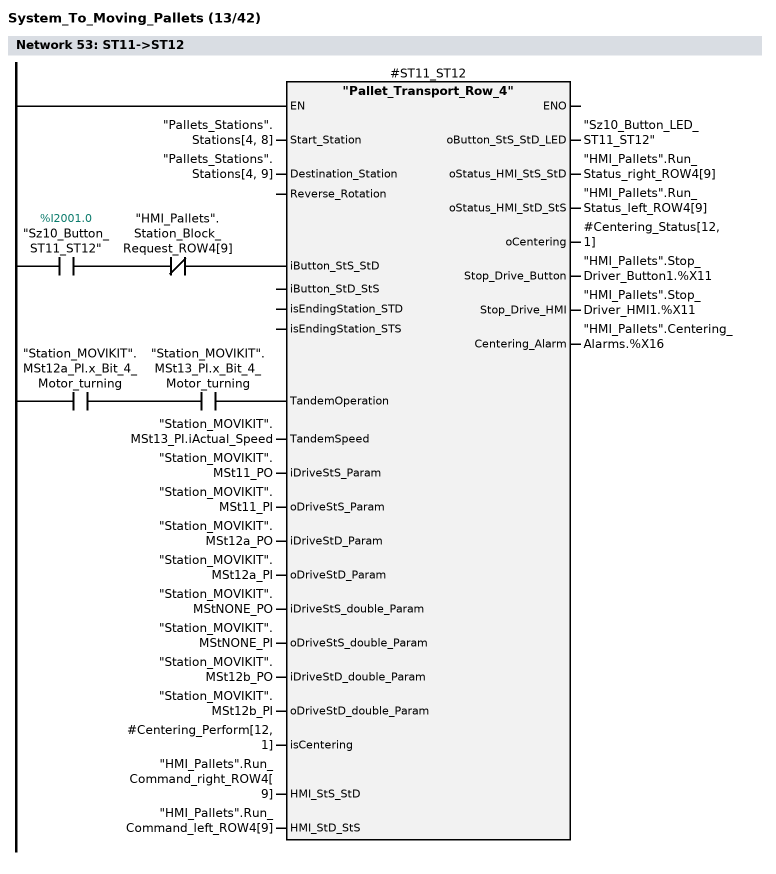
   RUNG wire#powerrail
      #ST11_ST12(iButton_StS_StD := wire#w1, TandemOperation := wire#w2, Start_Station := "Pallets_Stations".Stations[4, 8], Destination_Station := "Pallets_Stations".Stations[4, 9], Reverse_Rotation :=, iButton_StD_StS :=, isEndingStation_STD :=, isEndingStation_STS :=, TandemSpeed := "Station_MOVIKIT".MSt13_PI.iActual_Speed, iDriveStS_Param := "Station_MOVIKIT".MSt11_PO, oDriveStS_Param := "Station_MOVIKIT".MSt11_PI, iDriveStD_Param := "Station_MOVIKIT".MSt12a_PO, oDriveStD_Param := "Station_MOVIKIT".MSt12a_PI, iDriveStS_double_Param := "Station_MOVIKIT".MStNONE_PO, oDriveStS_double_Param := "Station_MOVIKIT".MStNONE_PI, iDriveStD_double_Param := "Station_MOVIKIT".MSt12b_PO, oDriveStD_double_Param := "Station_MOVIKIT".MSt12b_PI, isCentering := #Centering_Perform[12, 1], HMI_StS_StD := "HMI_Pallets".Run_Command_right_ROW4[9], HMI_StD_StS := "HMI_Pallets".Run_Command_left_ROW4[9], oButton_StS_StD_LED => "Sz10_Button_LED_ST11_ST12", oStatus_HMI_StS_StD => "HMI_Pallets".Run_Status_right_ROW4[9], oStatus_HMI_StD_StS => "HMI_Pallets".Run_Status_left_ROW4[9], oCentering => #Centering_Status[12, 1], Stop_Drive_Button => "HMI_Pallets".Stop_Driver_Button1.%X11, Stop_Drive_HMI => "HMI_Pallets".Stop_Driver_HMI1.%X11, Centering_Alarm => "HMI_Pallets".Centering_Alarms.%X16)
   END_RUNG
   RUNG wire#powerrail
      Contact( "Sz10_Button_ST11_ST12" )
      I_Contact( "HMI_Pallets".Station_Block_Request_ROW4[9] )
   END_RUNG wire#w1
   RUNG wire#powerrail
      Contact( "Station_MOVIKIT".MSt12a_PI.x_Bit_4_Motor_turning )
      Contact( "Station_MOVIKIT".MSt13_PI.x_Bit_4_Motor_turning )
   END_RUNG wire#w2
   // the same network as SCL:
   #ST11_ST12(Start_Station := "Pallets_Stations".Stations[4, 8],   // "Pallet_Transport_Row_4"
              Destination_Station := "Pallets_Stations".Stations[4, 9],
              iButton_StS_StD := "Sz10_Button_ST11_ST12" AND NOT "HMI_Pallets".Station_Block_Request_ROW4[9],
              TandemOperation := "Station_MOVIKIT".MSt12a_PI.x_Bit_4_Motor_turning AND "Station_MOVIKIT".MSt13_PI.x_Bit_4_Motor_turning,
              TandemSpeed := "Station_MOVIKIT".MSt13_PI.iActual_Speed,
              iDriveStS_Param := "Station_MOVIKIT".MSt11_PO,
              oDriveStS_Param := "Station_MOVIKIT".MSt11_PI,
              iDriveStD_Param := "Station_MOVIKIT".MSt12a_PO,
              oDriveStD_Param := "Station_MOVIKIT".MSt12a_PI,
              iDriveStS_double_Param := "Station_MOVIKIT".MStNONE_PO,
              oDriveStS_double_Param := "Station_MOVIKIT".MStNONE_PI,
              iDriveStD_double_Param := "Station_MOVIKIT".MSt12b_PO,
              oDriveStD_double_Param := "Station_MOVIKIT".MSt12b_PI,
              isCentering := #Centering_Perform[12, 1],
              HMI_StS_StD := "HMI_Pallets".Run_Command_right_ROW4[9],
              HMI_StD_StS := "HMI_Pallets".Run_Command_left_ROW4[9],
              oButton_StS_StD_LED => "Sz10_Button_LED_ST11_ST12",
              oStatus_HMI_StS_StD => "HMI_Pallets".Run_Status_right_ROW4[9],
              oStatus_HMI_StD_StS => "HMI_Pallets".Run_Status_left_ROW4[9],
              oCentering => #Centering_Status[12, 1],
              Stop_Drive_Button => "HMI_Pallets".Stop_Driver_Button1.%X11,
              Stop_Drive_HMI => "HMI_Pallets".Stop_Driver_HMI1.%X11,
              Centering_Alarm => "HMI_Pallets".Centering_Alarms.%X16);
END_REGION

REGION Network 54: ST10->ST11
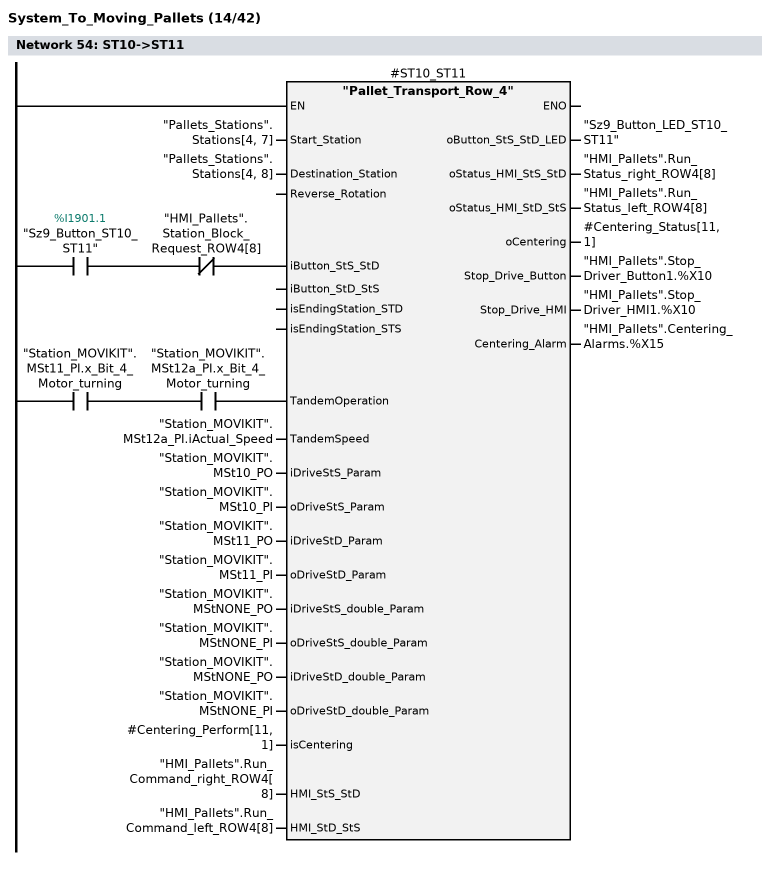
   RUNG wire#powerrail
      #ST10_ST11(iButton_StS_StD := wire#w1, TandemOperation := wire#w2, Start_Station := "Pallets_Stations".Stations[4, 7], Destination_Station := "Pallets_Stations".Stations[4, 8], Reverse_Rotation :=, iButton_StD_StS :=, isEndingStation_STD :=, isEndingStation_STS :=, TandemSpeed := "Station_MOVIKIT".MSt12a_PI.iActual_Speed, iDriveStS_Param := "Station_MOVIKIT".MSt10_PO, oDriveStS_Param := "Station_MOVIKIT".MSt10_PI, iDriveStD_Param := "Station_MOVIKIT".MSt11_PO, oDriveStD_Param := "Station_MOVIKIT".MSt11_PI, iDriveStS_double_Param := "Station_MOVIKIT".MStNONE_PO, oDriveStS_double_Param := "Station_MOVIKIT".MStNONE_PI, iDriveStD_double_Param := "Station_MOVIKIT".MStNONE_PO, oDriveStD_double_Param := "Station_MOVIKIT".MStNONE_PI, isCentering := #Centering_Perform[11, 1], HMI_StS_StD := "HMI_Pallets".Run_Command_right_ROW4[8], HMI_StD_StS := "HMI_Pallets".Run_Command_left_ROW4[8], oButton_StS_StD_LED => "Sz9_Button_LED_ST10_ST11", oStatus_HMI_StS_StD => "HMI_Pallets".Run_Status_right_ROW4[8], oStatus_HMI_StD_StS => "HMI_Pallets".Run_Status_left_ROW4[8], oCentering => #Centering_Status[11, 1], Stop_Drive_Button => "HMI_Pallets".Stop_Driver_Button1.%X10, Stop_Drive_HMI => "HMI_Pallets".Stop_Driver_HMI1.%X10, Centering_Alarm => "HMI_Pallets".Centering_Alarms.%X15)
   END_RUNG
   RUNG wire#powerrail
      Contact( "Sz9_Button_ST10_ST11" )
      I_Contact( "HMI_Pallets".Station_Block_Request_ROW4[8] )
   END_RUNG wire#w1
   RUNG wire#powerrail
      Contact( "Station_MOVIKIT".MSt11_PI.x_Bit_4_Motor_turning )
      Contact( "Station_MOVIKIT".MSt12a_PI.x_Bit_4_Motor_turning )
   END_RUNG wire#w2
   // the same network as SCL:
   #ST10_ST11(Start_Station := "Pallets_Stations".Stations[4, 7],   // "Pallet_Transport_Row_4"
              Destination_Station := "Pallets_Stations".Stations[4, 8],
              iButton_StS_StD := "Sz9_Button_ST10_ST11" AND NOT "HMI_Pallets".Station_Block_Request_ROW4[8],
              TandemOperation := "Station_MOVIKIT".MSt11_PI.x_Bit_4_Motor_turning AND "Station_MOVIKIT".MSt12a_PI.x_Bit_4_Motor_turning,
              TandemSpeed := "Station_MOVIKIT".MSt12a_PI.iActual_Speed,
              iDriveStS_Param := "Station_MOVIKIT".MSt10_PO,
              oDriveStS_Param := "Station_MOVIKIT".MSt10_PI,
              iDriveStD_Param := "Station_MOVIKIT".MSt11_PO,
              oDriveStD_Param := "Station_MOVIKIT".MSt11_PI,
              iDriveStS_double_Param := "Station_MOVIKIT".MStNONE_PO,
              oDriveStS_double_Param := "Station_MOVIKIT".MStNONE_PI,
              iDriveStD_double_Param := "Station_MOVIKIT".MStNONE_PO,
              oDriveStD_double_Param := "Station_MOVIKIT".MStNONE_PI,
              isCentering := #Centering_Perform[11, 1],
              HMI_StS_StD := "HMI_Pallets".Run_Command_right_ROW4[8],
              HMI_StD_StS := "HMI_Pallets".Run_Command_left_ROW4[8],
              oButton_StS_StD_LED => "Sz9_Button_LED_ST10_ST11",
              oStatus_HMI_StS_StD => "HMI_Pallets".Run_Status_right_ROW4[8],
              oStatus_HMI_StD_StS => "HMI_Pallets".Run_Status_left_ROW4[8],
              oCentering => #Centering_Status[11, 1],
              Stop_Drive_Button => "HMI_Pallets".Stop_Driver_Button1.%X10,
              Stop_Drive_HMI => "HMI_Pallets".Stop_Driver_HMI1.%X10,
              Centering_Alarm => "HMI_Pallets".Centering_Alarms.%X15);
END_REGION

REGION Network 55: ST09->ST10
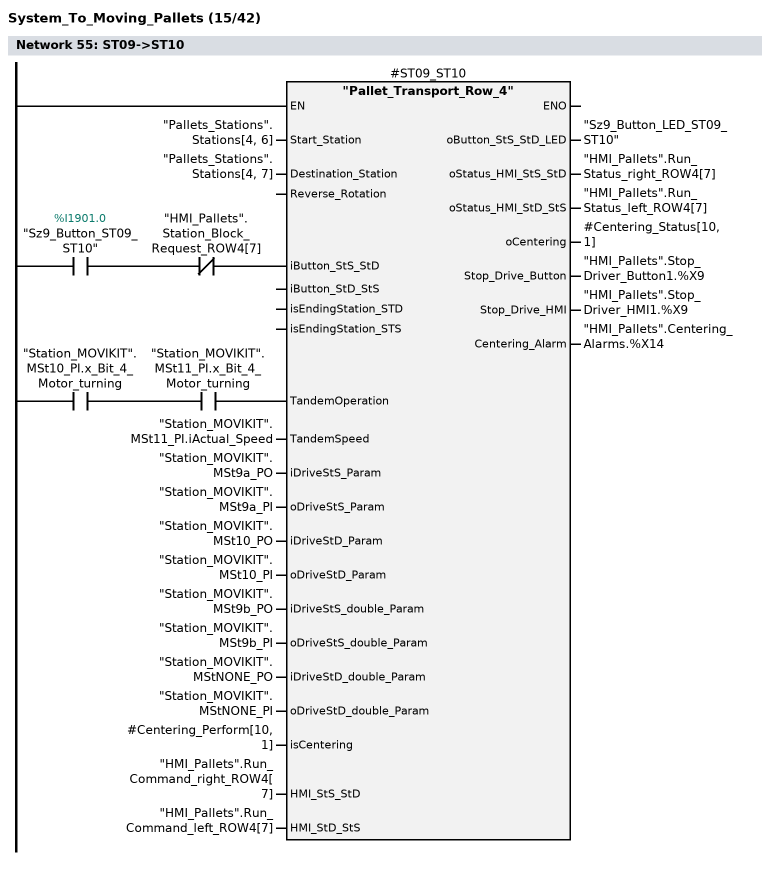
   RUNG wire#powerrail
      #ST09_ST10(iButton_StS_StD := wire#w1, TandemOperation := wire#w2, Start_Station := "Pallets_Stations".Stations[4, 6], Destination_Station := "Pallets_Stations".Stations[4, 7], Reverse_Rotation :=, iButton_StD_StS :=, isEndingStation_STD :=, isEndingStation_STS :=, TandemSpeed := "Station_MOVIKIT".MSt11_PI.iActual_Speed, iDriveStS_Param := "Station_MOVIKIT".MSt9a_PO, oDriveStS_Param := "Station_MOVIKIT".MSt9a_PI, iDriveStD_Param := "Station_MOVIKIT".MSt10_PO, oDriveStD_Param := "Station_MOVIKIT".MSt10_PI, iDriveStS_double_Param := "Station_MOVIKIT".MSt9b_PO, oDriveStS_double_Param := "Station_MOVIKIT".MSt9b_PI, iDriveStD_double_Param := "Station_MOVIKIT".MStNONE_PO, oDriveStD_double_Param := "Station_MOVIKIT".MStNONE_PI, isCentering := #Centering_Perform[10, 1], HMI_StS_StD := "HMI_Pallets".Run_Command_right_ROW4[7], HMI_StD_StS := "HMI_Pallets".Run_Command_left_ROW4[7], oButton_StS_StD_LED => "Sz9_Button_LED_ST09_ST10", oStatus_HMI_StS_StD => "HMI_Pallets".Run_Status_right_ROW4[7], oStatus_HMI_StD_StS => "HMI_Pallets".Run_Status_left_ROW4[7], oCentering => #Centering_Status[10, 1], Stop_Drive_Button => "HMI_Pallets".Stop_Driver_Button1.%X9, Stop_Drive_HMI => "HMI_Pallets".Stop_Driver_HMI1.%X9, Centering_Alarm => "HMI_Pallets".Centering_Alarms.%X14)
   END_RUNG
   RUNG wire#powerrail
      Contact( "Sz9_Button_ST09_ST10" )
      I_Contact( "HMI_Pallets".Station_Block_Request_ROW4[7] )
   END_RUNG wire#w1
   RUNG wire#powerrail
      Contact( "Station_MOVIKIT".MSt10_PI.x_Bit_4_Motor_turning )
      Contact( "Station_MOVIKIT".MSt11_PI.x_Bit_4_Motor_turning )
   END_RUNG wire#w2
   // the same network as SCL:
   #ST09_ST10(Start_Station := "Pallets_Stations".Stations[4, 6],   // "Pallet_Transport_Row_4"
              Destination_Station := "Pallets_Stations".Stations[4, 7],
              iButton_StS_StD := "Sz9_Button_ST09_ST10" AND NOT "HMI_Pallets".Station_Block_Request_ROW4[7],
              TandemOperation := "Station_MOVIKIT".MSt10_PI.x_Bit_4_Motor_turning AND "Station_MOVIKIT".MSt11_PI.x_Bit_4_Motor_turning,
              TandemSpeed := "Station_MOVIKIT".MSt11_PI.iActual_Speed,
              iDriveStS_Param := "Station_MOVIKIT".MSt9a_PO,
              oDriveStS_Param := "Station_MOVIKIT".MSt9a_PI,
              iDriveStD_Param := "Station_MOVIKIT".MSt10_PO,
              oDriveStD_Param := "Station_MOVIKIT".MSt10_PI,
              iDriveStS_double_Param := "Station_MOVIKIT".MSt9b_PO,
              oDriveStS_double_Param := "Station_MOVIKIT".MSt9b_PI,
              iDriveStD_double_Param := "Station_MOVIKIT".MStNONE_PO,
              oDriveStD_double_Param := "Station_MOVIKIT".MStNONE_PI,
              isCentering := #Centering_Perform[10, 1],
              HMI_StS_StD := "HMI_Pallets".Run_Command_right_ROW4[7],
              HMI_StD_StS := "HMI_Pallets".Run_Command_left_ROW4[7],
              oButton_StS_StD_LED => "Sz9_Button_LED_ST09_ST10",
              oStatus_HMI_StS_StD => "HMI_Pallets".Run_Status_right_ROW4[7],
              oStatus_HMI_StD_StS => "HMI_Pallets".Run_Status_left_ROW4[7],
              oCentering => #Centering_Status[10, 1],
              Stop_Drive_Button => "HMI_Pallets".Stop_Driver_Button1.%X9,
              Stop_Drive_HMI => "HMI_Pallets".Stop_Driver_HMI1.%X9,
              Centering_Alarm => "HMI_Pallets".Centering_Alarms.%X14);
END_REGION

REGION Network 56: ST08->ST09
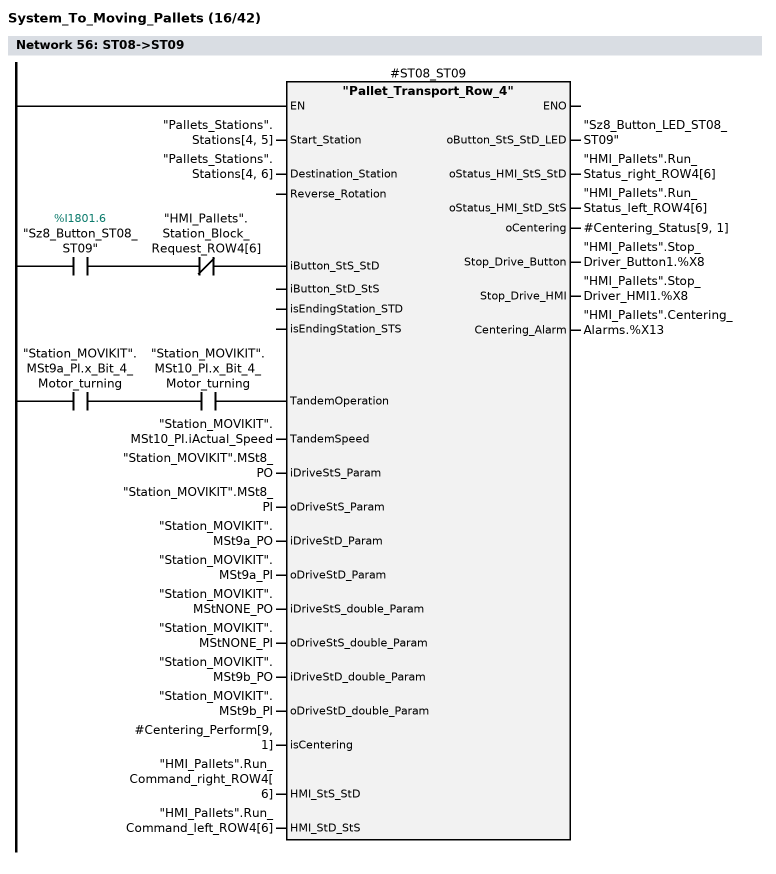
   RUNG wire#powerrail
      #ST08_ST09(iButton_StS_StD := wire#w1, TandemOperation := wire#w2, Start_Station := "Pallets_Stations".Stations[4, 5], Destination_Station := "Pallets_Stations".Stations[4, 6], Reverse_Rotation :=, iButton_StD_StS :=, isEndingStation_STD :=, isEndingStation_STS :=, TandemSpeed := "Station_MOVIKIT".MSt10_PI.iActual_Speed, iDriveStS_Param := "Station_MOVIKIT".MSt8_PO, oDriveStS_Param := "Station_MOVIKIT".MSt8_PI, iDriveStD_Param := "Station_MOVIKIT".MSt9a_PO, oDriveStD_Param := "Station_MOVIKIT".MSt9a_PI, iDriveStS_double_Param := "Station_MOVIKIT".MStNONE_PO, oDriveStS_double_Param := "Station_MOVIKIT".MStNONE_PI, iDriveStD_double_Param := "Station_MOVIKIT".MSt9b_PO, oDriveStD_double_Param := "Station_MOVIKIT".MSt9b_PI, isCentering := #Centering_Perform[9, 1], HMI_StS_StD := "HMI_Pallets".Run_Command_right_ROW4[6], HMI_StD_StS := "HMI_Pallets".Run_Command_left_ROW4[6], oButton_StS_StD_LED => "Sz8_Button_LED_ST08_ST09", oStatus_HMI_StS_StD => "HMI_Pallets".Run_Status_right_ROW4[6], oStatus_HMI_StD_StS => "HMI_Pallets".Run_Status_left_ROW4[6], oCentering => #Centering_Status[9, 1], Stop_Drive_Button => "HMI_Pallets".Stop_Driver_Button1.%X8, Stop_Drive_HMI => "HMI_Pallets".Stop_Driver_HMI1.%X8, Centering_Alarm => "HMI_Pallets".Centering_Alarms.%X13)
   END_RUNG
   RUNG wire#powerrail
      Contact( "Sz8_Button_ST08_ST09" )
      I_Contact( "HMI_Pallets".Station_Block_Request_ROW4[6] )
   END_RUNG wire#w1
   RUNG wire#powerrail
      Contact( "Station_MOVIKIT".MSt9a_PI.x_Bit_4_Motor_turning )
      Contact( "Station_MOVIKIT".MSt10_PI.x_Bit_4_Motor_turning )
   END_RUNG wire#w2
   // the same network as SCL:
   #ST08_ST09(Start_Station := "Pallets_Stations".Stations[4, 5],   // "Pallet_Transport_Row_4"
              Destination_Station := "Pallets_Stations".Stations[4, 6],
              iButton_StS_StD := "Sz8_Button_ST08_ST09" AND NOT "HMI_Pallets".Station_Block_Request_ROW4[6],
              TandemOperation := "Station_MOVIKIT".MSt9a_PI.x_Bit_4_Motor_turning AND "Station_MOVIKIT".MSt10_PI.x_Bit_4_Motor_turning,
              TandemSpeed := "Station_MOVIKIT".MSt10_PI.iActual_Speed,
              iDriveStS_Param := "Station_MOVIKIT".MSt8_PO,
              oDriveStS_Param := "Station_MOVIKIT".MSt8_PI,
              iDriveStD_Param := "Station_MOVIKIT".MSt9a_PO,
              oDriveStD_Param := "Station_MOVIKIT".MSt9a_PI,
              iDriveStS_double_Param := "Station_MOVIKIT".MStNONE_PO,
              oDriveStS_double_Param := "Station_MOVIKIT".MStNONE_PI,
              iDriveStD_double_Param := "Station_MOVIKIT".MSt9b_PO,
              oDriveStD_double_Param := "Station_MOVIKIT".MSt9b_PI,
              isCentering := #Centering_Perform[9, 1],
              HMI_StS_StD := "HMI_Pallets".Run_Command_right_ROW4[6],
              HMI_StD_StS := "HMI_Pallets".Run_Command_left_ROW4[6],
              oButton_StS_StD_LED => "Sz8_Button_LED_ST08_ST09",
              oStatus_HMI_StS_StD => "HMI_Pallets".Run_Status_right_ROW4[6],
              oStatus_HMI_StD_StS => "HMI_Pallets".Run_Status_left_ROW4[6],
              oCentering => #Centering_Status[9, 1],
              Stop_Drive_Button => "HMI_Pallets".Stop_Driver_Button1.%X8,
              Stop_Drive_HMI => "HMI_Pallets".Stop_Driver_HMI1.%X8,
              Centering_Alarm => "HMI_Pallets".Centering_Alarms.%X13);
END_REGION

REGION Network 57: ST07->ST08
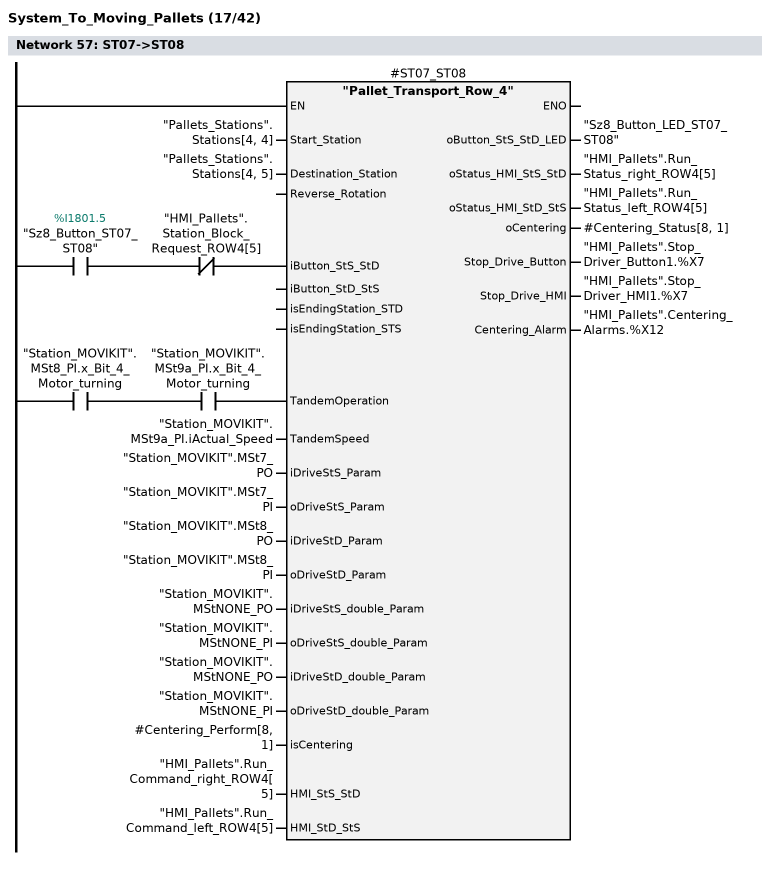
   RUNG wire#powerrail
      #ST07_ST08(iButton_StS_StD := wire#w1, TandemOperation := wire#w2, Start_Station := "Pallets_Stations".Stations[4, 4], Destination_Station := "Pallets_Stations".Stations[4, 5], Reverse_Rotation :=, iButton_StD_StS :=, isEndingStation_STD :=, isEndingStation_STS :=, TandemSpeed := "Station_MOVIKIT".MSt9a_PI.iActual_Speed, iDriveStS_Param := "Station_MOVIKIT".MSt7_PO, oDriveStS_Param := "Station_MOVIKIT".MSt7_PI, iDriveStD_Param := "Station_MOVIKIT".MSt8_PO, oDriveStD_Param := "Station_MOVIKIT".MSt8_PI, iDriveStS_double_Param := "Station_MOVIKIT".MStNONE_PO, oDriveStS_double_Param := "Station_MOVIKIT".MStNONE_PI, iDriveStD_double_Param := "Station_MOVIKIT".MStNONE_PO, oDriveStD_double_Param := "Station_MOVIKIT".MStNONE_PI, isCentering := #Centering_Perform[8, 1], HMI_StS_StD := "HMI_Pallets".Run_Command_right_ROW4[5], HMI_StD_StS := "HMI_Pallets".Run_Command_left_ROW4[5], oButton_StS_StD_LED => "Sz8_Button_LED_ST07_ST08", oStatus_HMI_StS_StD => "HMI_Pallets".Run_Status_right_ROW4[5], oStatus_HMI_StD_StS => "HMI_Pallets".Run_Status_left_ROW4[5], oCentering => #Centering_Status[8, 1], Stop_Drive_Button => "HMI_Pallets".Stop_Driver_Button1.%X7, Stop_Drive_HMI => "HMI_Pallets".Stop_Driver_HMI1.%X7, Centering_Alarm => "HMI_Pallets".Centering_Alarms.%X12)
   END_RUNG
   RUNG wire#powerrail
      Contact( "Sz8_Button_ST07_ST08" )
      I_Contact( "HMI_Pallets".Station_Block_Request_ROW4[5] )
   END_RUNG wire#w1
   RUNG wire#powerrail
      Contact( "Station_MOVIKIT".MSt8_PI.x_Bit_4_Motor_turning )
      Contact( "Station_MOVIKIT".MSt9a_PI.x_Bit_4_Motor_turning )
   END_RUNG wire#w2
   // the same network as SCL:
   #ST07_ST08(Start_Station := "Pallets_Stations".Stations[4, 4],   // "Pallet_Transport_Row_4"
              Destination_Station := "Pallets_Stations".Stations[4, 5],
              iButton_StS_StD := "Sz8_Button_ST07_ST08" AND NOT "HMI_Pallets".Station_Block_Request_ROW4[5],
              TandemOperation := "Station_MOVIKIT".MSt8_PI.x_Bit_4_Motor_turning AND "Station_MOVIKIT".MSt9a_PI.x_Bit_4_Motor_turning,
              TandemSpeed := "Station_MOVIKIT".MSt9a_PI.iActual_Speed,
              iDriveStS_Param := "Station_MOVIKIT".MSt7_PO,
              oDriveStS_Param := "Station_MOVIKIT".MSt7_PI,
              iDriveStD_Param := "Station_MOVIKIT".MSt8_PO,
              oDriveStD_Param := "Station_MOVIKIT".MSt8_PI,
              iDriveStS_double_Param := "Station_MOVIKIT".MStNONE_PO,
              oDriveStS_double_Param := "Station_MOVIKIT".MStNONE_PI,
              iDriveStD_double_Param := "Station_MOVIKIT".MStNONE_PO,
              oDriveStD_double_Param := "Station_MOVIKIT".MStNONE_PI,
              isCentering := #Centering_Perform[8, 1],
              HMI_StS_StD := "HMI_Pallets".Run_Command_right_ROW4[5],
              HMI_StD_StS := "HMI_Pallets".Run_Command_left_ROW4[5],
              oButton_StS_StD_LED => "Sz8_Button_LED_ST07_ST08",
              oStatus_HMI_StS_StD => "HMI_Pallets".Run_Status_right_ROW4[5],
              oStatus_HMI_StD_StS => "HMI_Pallets".Run_Status_left_ROW4[5],
              oCentering => #Centering_Status[8, 1],
              Stop_Drive_Button => "HMI_Pallets".Stop_Driver_Button1.%X7,
              Stop_Drive_HMI => "HMI_Pallets".Stop_Driver_HMI1.%X7,
              Centering_Alarm => "HMI_Pallets".Centering_Alarms.%X12);
END_REGION

REGION Network 58: ST06->ST07
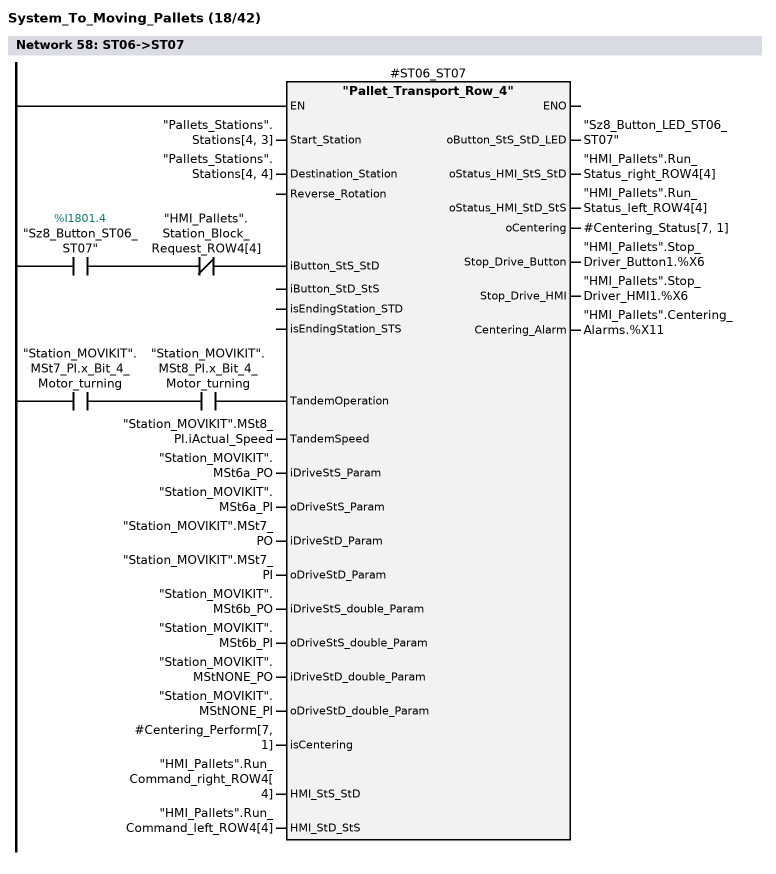
   RUNG wire#powerrail
      #ST06_ST07(iButton_StS_StD := wire#w1, TandemOperation := wire#w2, Start_Station := "Pallets_Stations".Stations[4, 3], Destination_Station := "Pallets_Stations".Stations[4, 4], Reverse_Rotation :=, iButton_StD_StS :=, isEndingStation_STD :=, isEndingStation_STS :=, TandemSpeed := "Station_MOVIKIT".MSt8_PI.iActual_Speed, iDriveStS_Param := "Station_MOVIKIT".MSt6a_PO, oDriveStS_Param := "Station_MOVIKIT".MSt6a_PI, iDriveStD_Param := "Station_MOVIKIT".MSt7_PO, oDriveStD_Param := "Station_MOVIKIT".MSt7_PI, iDriveStS_double_Param := "Station_MOVIKIT".MSt6b_PO, oDriveStS_double_Param := "Station_MOVIKIT".MSt6b_PI, iDriveStD_double_Param := "Station_MOVIKIT".MStNONE_PO, oDriveStD_double_Param := "Station_MOVIKIT".MStNONE_PI, isCentering := #Centering_Perform[7, 1], HMI_StS_StD := "HMI_Pallets".Run_Command_right_ROW4[4], HMI_StD_StS := "HMI_Pallets".Run_Command_left_ROW4[4], oButton_StS_StD_LED => "Sz8_Button_LED_ST06_ST07", oStatus_HMI_StS_StD => "HMI_Pallets".Run_Status_right_ROW4[4], oStatus_HMI_StD_StS => "HMI_Pallets".Run_Status_left_ROW4[4], oCentering => #Centering_Status[7, 1], Stop_Drive_Button => "HMI_Pallets".Stop_Driver_Button1.%X6, Stop_Drive_HMI => "HMI_Pallets".Stop_Driver_HMI1.%X6, Centering_Alarm => "HMI_Pallets".Centering_Alarms.%X11)
   END_RUNG
   RUNG wire#powerrail
      Contact( "Sz8_Button_ST06_ST07" )
      I_Contact( "HMI_Pallets".Station_Block_Request_ROW4[4] )
   END_RUNG wire#w1
   RUNG wire#powerrail
      Contact( "Station_MOVIKIT".MSt7_PI.x_Bit_4_Motor_turning )
      Contact( "Station_MOVIKIT".MSt8_PI.x_Bit_4_Motor_turning )
   END_RUNG wire#w2
   // the same network as SCL:
   #ST06_ST07(Start_Station := "Pallets_Stations".Stations[4, 3],   // "Pallet_Transport_Row_4"
              Destination_Station := "Pallets_Stations".Stations[4, 4],
              iButton_StS_StD := "Sz8_Button_ST06_ST07" AND NOT "HMI_Pallets".Station_Block_Request_ROW4[4],
              TandemOperation := "Station_MOVIKIT".MSt7_PI.x_Bit_4_Motor_turning AND "Station_MOVIKIT".MSt8_PI.x_Bit_4_Motor_turning,
              TandemSpeed := "Station_MOVIKIT".MSt8_PI.iActual_Speed,
              iDriveStS_Param := "Station_MOVIKIT".MSt6a_PO,
              oDriveStS_Param := "Station_MOVIKIT".MSt6a_PI,
              iDriveStD_Param := "Station_MOVIKIT".MSt7_PO,
              oDriveStD_Param := "Station_MOVIKIT".MSt7_PI,
              iDriveStS_double_Param := "Station_MOVIKIT".MSt6b_PO,
              oDriveStS_double_Param := "Station_MOVIKIT".MSt6b_PI,
              iDriveStD_double_Param := "Station_MOVIKIT".MStNONE_PO,
              oDriveStD_double_Param := "Station_MOVIKIT".MStNONE_PI,
              isCentering := #Centering_Perform[7, 1],
              HMI_StS_StD := "HMI_Pallets".Run_Command_right_ROW4[4],
              HMI_StD_StS := "HMI_Pallets".Run_Command_left_ROW4[4],
              oButton_StS_StD_LED => "Sz8_Button_LED_ST06_ST07",
              oStatus_HMI_StS_StD => "HMI_Pallets".Run_Status_right_ROW4[4],
              oStatus_HMI_StD_StS => "HMI_Pallets".Run_Status_left_ROW4[4],
              oCentering => #Centering_Status[7, 1],
              Stop_Drive_Button => "HMI_Pallets".Stop_Driver_Button1.%X6,
              Stop_Drive_HMI => "HMI_Pallets".Stop_Driver_HMI1.%X6,
              Centering_Alarm => "HMI_Pallets".Centering_Alarms.%X11);
END_REGION

REGION Network 59: ST05->ST06
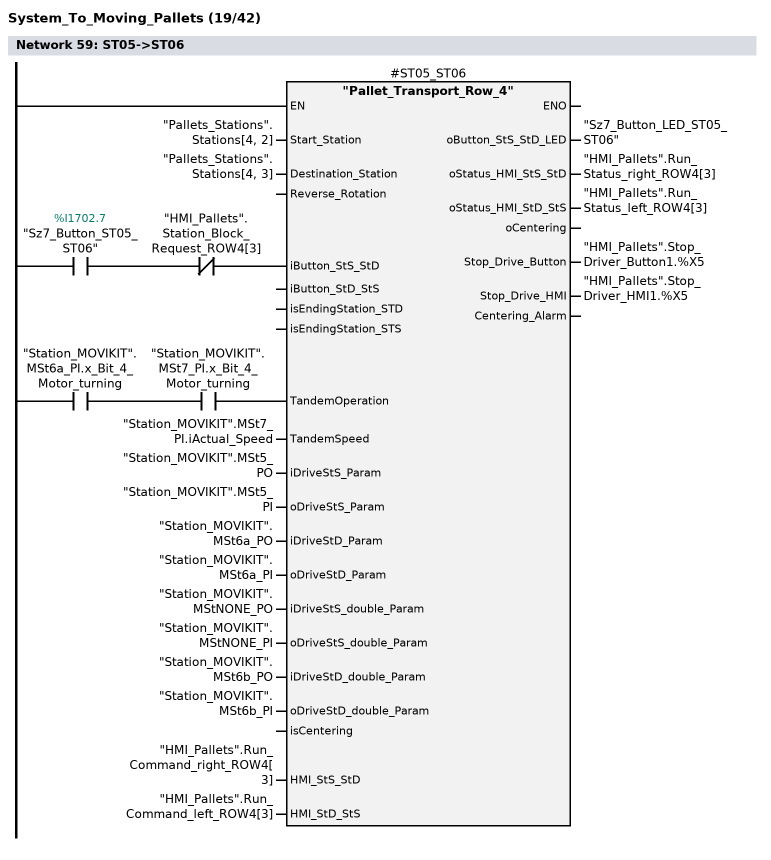
   RUNG wire#powerrail
      #ST05_ST06(iButton_StS_StD := wire#w1, TandemOperation := wire#w2, Start_Station := "Pallets_Stations".Stations[4, 2], Destination_Station := "Pallets_Stations".Stations[4, 3], Reverse_Rotation :=, iButton_StD_StS :=, isEndingStation_STD :=, isEndingStation_STS :=, TandemSpeed := "Station_MOVIKIT".MSt7_PI.iActual_Speed, iDriveStS_Param := "Station_MOVIKIT".MSt5_PO, oDriveStS_Param := "Station_MOVIKIT".MSt5_PI, iDriveStD_Param := "Station_MOVIKIT".MSt6a_PO, oDriveStD_Param := "Station_MOVIKIT".MSt6a_PI, iDriveStS_double_Param := "Station_MOVIKIT".MStNONE_PO, oDriveStS_double_Param := "Station_MOVIKIT".MStNONE_PI, iDriveStD_double_Param := "Station_MOVIKIT".MSt6b_PO, oDriveStD_double_Param := "Station_MOVIKIT".MSt6b_PI, isCentering :=, HMI_StS_StD := "HMI_Pallets".Run_Command_right_ROW4[3], HMI_StD_StS := "HMI_Pallets".Run_Command_left_ROW4[3], oButton_StS_StD_LED => "Sz7_Button_LED_ST05_ST06", oStatus_HMI_StS_StD => "HMI_Pallets".Run_Status_right_ROW4[3], oStatus_HMI_StD_StS => "HMI_Pallets".Run_Status_left_ROW4[3], oCentering =>, Stop_Drive_Button => "HMI_Pallets".Stop_Driver_Button1.%X5, Stop_Drive_HMI => "HMI_Pallets".Stop_Driver_HMI1.%X5, Centering_Alarm =>)
   END_RUNG
   RUNG wire#powerrail
      Contact( "Sz7_Button_ST05_ST06" )
      I_Contact( "HMI_Pallets".Station_Block_Request_ROW4[3] )
   END_RUNG wire#w1
   RUNG wire#powerrail
      Contact( "Station_MOVIKIT".MSt6a_PI.x_Bit_4_Motor_turning )
      Contact( "Station_MOVIKIT".MSt7_PI.x_Bit_4_Motor_turning )
   END_RUNG wire#w2
   // the same network as SCL:
   #ST05_ST06(Start_Station := "Pallets_Stations".Stations[4, 2],   // "Pallet_Transport_Row_4"
              Destination_Station := "Pallets_Stations".Stations[4, 3],
              iButton_StS_StD := "Sz7_Button_ST05_ST06" AND NOT "HMI_Pallets".Station_Block_Request_ROW4[3],
              TandemOperation := "Station_MOVIKIT".MSt6a_PI.x_Bit_4_Motor_turning AND "Station_MOVIKIT".MSt7_PI.x_Bit_4_Motor_turning,
              TandemSpeed := "Station_MOVIKIT".MSt7_PI.iActual_Speed,
              iDriveStS_Param := "Station_MOVIKIT".MSt5_PO,
              oDriveStS_Param := "Station_MOVIKIT".MSt5_PI,
              iDriveStD_Param := "Station_MOVIKIT".MSt6a_PO,
              oDriveStD_Param := "Station_MOVIKIT".MSt6a_PI,
              iDriveStS_double_Param := "Station_MOVIKIT".MStNONE_PO,
              oDriveStS_double_Param := "Station_MOVIKIT".MStNONE_PI,
              iDriveStD_double_Param := "Station_MOVIKIT".MSt6b_PO,
              oDriveStD_double_Param := "Station_MOVIKIT".MSt6b_PI,
              HMI_StS_StD := "HMI_Pallets".Run_Command_right_ROW4[3],
              HMI_StD_StS := "HMI_Pallets".Run_Command_left_ROW4[3],
              oButton_StS_StD_LED => "Sz7_Button_LED_ST05_ST06",
              oStatus_HMI_StS_StD => "HMI_Pallets".Run_Status_right_ROW4[3],
              oStatus_HMI_StD_StS => "HMI_Pallets".Run_Status_left_ROW4[3],
              Stop_Drive_Button => "HMI_Pallets".Stop_Driver_Button1.%X5,
              Stop_Drive_HMI => "HMI_Pallets".Stop_Driver_HMI1.%X5);
END_REGION

